IF NOT(xReadFirstTime) THEN
	xReadFirstTime:=TRUE;
END_IF;
(******************************************************************************************************************************************)
(****************************				           Reset Function Part                                                 *****************************)
(******************************************************************************************************************************************)
IF xReset AND NOT(xSetEnd) THEN
	xEnd:=FALSE;
	xSetEnd:=TRUE;
END_IF;
(******************************************************************************************************************************************)
(****************************				              Error Controlling Part                                            *****************************)
(******************************************************************************************************************************************)
xTmp:=	TAxisToolLeft.T_CtrleSingle.xErr OR
		(TAxisToolCenter.T_CtrleSingle.xErr AND xMicroRodActive) OR
		TAxisToolRight.T_CtrleSingle.xErr OR
		TAxisToolFeeder.T_CtrleSingle.xErr OR
		TAxisGrindFeeder.T_CtrleSingle.xErr;
xTmp1:=	NOT(TAxisToolLeft.T_CtrleSingle.xExecute) AND
		((NOT(TAxisToolCenter.T_CtrleSingle.xExecute) AND xMicroRodActive) OR NOT(xMicroRodActive)) AND
		 NOT(TAxisToolRight.T_CtrleSingle.xExecute) AND
		((NOT(TAxisToolFeeder.T_CtrleSingle.xExecute) AND NOT(xMicroRodActive)) OR xMicroRodActive) AND
		NOT(TAxisGrindFeeder.T_CtrleSingle.xExecute);
IF (xHardwareError OR (xTmp AND xStartMainPrc)) AND NOT(xSetEnd) THEN
	IF xTmp1 THEN
		IF NOT(xInitError) THEN
			iStepError:=100;
			xInitError:=TRUE;
			IF xHardwareError THEN
				iErrorNr:=iTmpErrorNr;
			ELSE
				xHardwareError:=TRUE;	(* Hardware Error *)
			END_IF;
		END_IF;
		CASE iStepError OF
			100:	iStepError:=0;
				xError:=TRUE;
		END_CASE;
		IF xQuitErr THEN
			xSetEnd:=TRUE;
		END_IF;
	END_IF;
END_IF;
(******************************************************************************************************************************************)
(****************************				              Main Controlling Part                                            *****************************)
(******************************************************************************************************************************************)
IF (xStart OR xStartMainCtr) AND NOT(xSetEnd) AND NOT(xHardwareError) THEN
	IF NOT (xInitMainCtr) THEN
		iTmpErrorNr:=0;
		iStepPrc:=100;
		xInitMainCtr:=TRUE;
		xStartMainCtr:=TRUE;
		xStart:=FALSE;
		xEnd:=FALSE;
		xAbord:=FALSE;
		xTmpInit:=FALSE;
		xCheckToolFeedPosition:=FALSE;
		xCheckWithoutToolRotation:=FALSE;
		bActivePartNumber:=0;
		lrCalcToolLengthInc:=lrCalcToolLength:=0.0;
		rSpeedToolFeed:=0.0;
	END_IF;
	IF xStop AND NOT(xTmpInit) THEN
		xTmpInit:=TRUE;
		iTmp:=100;
		RETURN;
	END_IF;
	IF xFreeze THEN
		IF xStart AND NOT(xAbord) THEN
			xFreeze:=FALSE;
			xStart:=FALSE;
		END_IF;
		IF xAbord THEN
			xAbord:=FALSE;
			xFreeze:=FALSE;
			xStart:=FALSE;
			xSetEnd:=TRUE;
		END_IF;
		RETURN;
	END_IF;
	IF NOT(xStartMainPrc) AND NOT(xSetEnd) THEN
		xStartMainPrc:=TRUE;
	END_IF;
END_IF;
(******************************************************************************************************************************************)
(****************************		               Controlling of the ToolFeeder Position                            *****************************)
(******************************************************************************************************************************************)
IF xCheckToolFeedPosition THEN
	IF xMicroRodActive THEN
		lrToolFeederPosition:=TAxisToolFeeder.T_LiveValue.lrActualPositionNotModulo - lrSaveToolFeederPosition;
		lrToolFeederActualPosition:=(lrToolFeederPosition / TAxisToolFeeder.T_CtrleSingle.lrScaleFactor);
		lrCalcToolLength:=lrToolFeederActualPosition;
	END_IF;
	IF NOT(xMicroRodActive) AND (TAxisToolRight.T_CtrleSingle.lrGearRatio <> 0.0) THEN
		IF NOT(xCheckWithoutToolRotation) THEN
			lrToolFeedCalcLengthPosition:=((((T_WorkTool.rToolLength * 10.0) / ABS(T_WorkTool.rPitch)) * 24000.0) / TAxisToolRight.T_CtrleSingle.lrScaleFactor);
			lrToolFeederPosition:=lrToolFeederPosition + ABS(ABS(TAxisToolRight.T_LiveValue.lrActualPosition) - (lrSaveToolFeederPosition / TAxisToolRight.T_CtrleSingle.lrScaleFactor));
			lrSaveToolFeederPosition:=ABS(TAxisToolRight.T_LiveValue.lrActualPositionNotModulo);
			lrToolFeederActualPosition:=((T_WorkTool.rToolLength * 10.0) / lrToolFeedCalcLengthPosition) * lrToolFeederPosition;
			lrCalcToolLength:=lrCalcToolLengthInc + lrToolFeederActualPosition;
		ELSE
			lrCalcToolLength:=ABS(TAxisToolFeeder.T_LiveValue.lrActualPosition);
		END_IF;
	END_IF;
ELSE
	xCheckWithoutToolRotation:=FALSE;
	IF NOT(xMicroRodActive) AND (TAxisToolRight.T_CtrleSingle.lrGearRatio <> 0.0) THEN
		lrSaveToolFeederPosition:=ABS(TAxisToolRight.T_LiveValue.lrActualPositionNotModulo);
		lrSaveToolRightPosition:=TAxisToolRight.T_LiveValue.lrActualPositionNotModulo * TAxisToolRight.T_CtrleSingle.lrGearRatio;
		lrCalcToolLengthInc:=lrCalcToolLength;
	END_IF;
	IF xMicroRodActive THEN
		lrSaveToolFeederPosition:=TAxisToolFeeder.T_LiveValue.lrActualPositionNotModulo;
	END_IF;
	lrToolFeederActualPosition:=lrToolFeederPosition:=0.0;
END_IF;
lrProcessToolFeederActualPosition:=lrCalcToolLength;
lrProcessToolFeederSpeed:=rSpeedToolFeed;
(******************************************************************************************************************************************)
(****************************				             immediate Stop Part                                              *****************************)
(******************************************************************************************************************************************)
IF xTmpInit AND NOT(xSetEnd) THEN
	IF NOT(xSafetyCircuitOn) THEN
		xTmpInit:=FALSE;
		iTmp:=100;
		xSetEnd:=TRUE;
		RETURN;
	END_IF;
	CASE iTmp OF
		100:	xReadyToolFeedStop:=xReadyGrindFeedStop:=FALSE;
			TAxisGrindFeeder.T_CtrleSingle.lrAcceleration:=T_Standard.T_TeachINToolFeeder.rAcceleration;
			TAxisGrindFeeder.T_CtrleSingle.lrDecceleration:=T_Standard.T_TeachINToolFeeder.rDeceleration;
			TAxisGrindFeeder.T_CtrleSingle.iFunction:=5;	(* Stop Movement *)
			TAxisGrindFeeder.T_CtrleSingle.xExecute:=TRUE;
			iTmp:=200;
			RETURN;
		200:	IF NOT(TAxisGrindFeeder.T_CtrleSingle.xExecute) AND TAxisGrindFeeder.T_CtrleSingle.xDone THEN
				TAxisGrindFeeder.T_CtrleSingle.lrAcceleration:=T_Standard.T_TeachINGrindFeeder.rAcceleration;
				TAxisGrindFeeder.T_CtrleSingle.lrDecceleration:=T_Standard.T_TeachINGrindFeeder.rDeceleration;
				TAxisGrindFeeder.T_CtrleSingle.lrPosition:=	T_ProcessImageData.T_ProcessPara.rToolDiameterProcess +
														T_ProcessImageData.T_ProcessPara.rSecurityPosGrindFeedProcess;
				TAxisGrindFeeder.T_CtrleSingle.lrVelocity:=T_ProcessImageData.T_ProcessPara.rSpeedBackwardGrindFeed;
				TAxisGrindFeeder.T_CtrleSingle.iFunction:=7;	(* Move Absolut *)
				TAxisGrindFeeder.T_CtrleSingle.xExecute:=TRUE;
				iTmp:=300;
			END_IF;
			RETURN;
		300:	IF NOT(TAxisGrindFeeder.T_CtrleSingle.xExecute) AND TAxisGrindFeeder.T_CtrleSingle.xDone AND NOT(xReadyGrindFeedStop) THEN
				xReadyGrindFeedStop:=TRUE;
			END_IF;
			IF (TAxisGrindFeeder.T_LiveValue.lrActualPosition >= (T_ProcessImageData.T_ProcessPara.rToolDiameterProcess + T_ProcessImageData.T_ProcessPara.rOffsetBeforeToolDiaGrindFeedProcess)) AND NOT(xReadyToolFeedStop) THEN
				xReadyToolFeedStop:=TRUE;
				xCheckToolFeedPosition:=FALSE;
				IF xMicroRodActive THEN
					IF NOT(TAxisToolFeeder.T_CtrleSingle.xNotMoving) THEN
						TAxisToolFeeder.T_CtrleSingle.lrAcceleration:=T_Standard.T_TeachINToolFeeder.rAcceleration;
						TAxisToolFeeder.T_CtrleSingle.lrDecceleration:=T_Standard.T_TeachINToolFeeder.rDeceleration;
						TAxisToolFeeder.T_CtrleSingle.iFunction:=5;	(* Stop Movement *)
						TAxisToolFeeder.T_CtrleSingle.xExecute:=TRUE;
					END_IF;
				END_IF;
				IF NOT(xMicroRodActive) THEN
					FBCalcGearFactor(	rSpeed:= 0.0,
										rToolRotationSpeed:= rToolRotationSpeed,
										T_WorkTool:=T_WorkTool );
					IF (T_WorkTool.rToolRotationSpeed > 0) THEN
						TAxisToolFeeder.T_CtrleSingle.lrGearFactor:=INT_TO_LREAL(FBCalcGearFactor.T_WorkTool.iToolFeederGearFactor) * -1.0;
					ELSE
						TAxisToolFeeder.T_CtrleSingle.lrGearFactor:=INT_TO_LREAL(FBCalcGearFactor.T_WorkTool.iToolFeederGearFactor);
					END_IF;
					TAxisToolFeeder.T_CtrleSingle.lrGearDivider:=INT_TO_LREAL(FBCalcGearFactor.T_WorkTool.iToolFeederGearDivider);
					(* Set Gear Value with PDO Object *)
					TAxisToolFeeder.T_RxPdoParameter.iGearFactor:=LREAL_TO_INT(TAxisToolFeeder.T_CtrleSingle.lrGearFactor);
					TAxisToolFeeder.T_RxPdoParameter.uiGearDivider:=LREAL_TO_UINT(TAxisToolFeeder.T_CtrleSingle.lrGearDivider);
				END_IF;
				lrProcessToolFeederSpeed:=0.0;
			END_IF;
			IF xReadyToolFeedStop AND xReadyGrindFeedStop THEN
				iTmp:=400;
			END_IF;
			RETURN;
		400:	IF NOT(TAxisToolFeeder.T_CtrleSingle.xExecute) AND TAxisToolFeeder.T_CtrleSingle.xDone THEN
				iTmp:=500;
			END_IF;
			RETURN;
		500:	xTmpInit:=FALSE;
			iTmp:=100;
			xSetEnd:=TRUE;
			RETURN;
	END_CASE;
END_IF;
(******************************************************************************************************************************************)
(****************************				             Main Procedure Part                                             *****************************)
(******************************************************************************************************************************************)
IF xStartMainPrc AND NOT(xSetEnd) AND NOT(xHardwareError) THEN
	CASE iStepPrc OF
		(* Initial Procedure *)
		100:	rToolFeedLength:=0.0;
			rToolDiameter:=T_ProcessImageData.T_ProcessPara.rToolDiameterProcess;
			rGrindFeedPlunge:=0.0;
			rSpeedGrindFeed:=0.0;
			rSpeedToolFeed:=0.0;
			iStartSection:=1;
			(* Check Start and End Section of the ToolGeometry *)
			FOR ii:=1 TO 6 DO
				IF T_ProcessImageData.T_GeometryPara.axActiveSection[ii] THEN
					IF (iStartSection = 0) THEN
						iStartSection:=ii;
					END_IF;
					iEndSection:=ii;
				END_IF;
			END_FOR;
			xResetFB:=TRUE;
			FBCalcPlungeGrinding(	rToolDiameter:= T_ProcessImageData.T_ProcessPara.rToolDiameterProcess,
									rToolDiameterWithOffset:=T_ProcessImageData.T_ProcessPara.rToolDiameterProcess + T_ProcessImageData.T_ProcessPara.rOffsetBeforeToolDiaGrindFeedProcess,
									xReset:= xResetFB);
			(* AutoGroove is not aloved to work in more cycle *)
			rPlungeCycleGrindFeedGeometry:=T_ProcessImageData.T_ProcessPara.rToolDiameterProcess;
			xStartMainPrc:=FALSE;
			xInitStep:=FALSE;
(*08.09.2010: KFS	{ *)
(*			iStepPrc:=200;*)
			iStepPrc:=120;
		(* Switch the Axis as Slave for Move ToolRotation to StartPositionGroove*)
		120:	IF NOT(xInitStep) THEN
				xInitStep:=TRUE;
				IF rStartPosAutoGrooveToolRotation<> 0 THEN
					IF NOT(TAxisToolCenter.T_CtrleSingle.xSlave) THEN
						TAxisToolCenter.T_CtrleSingle.lrGearDivider:=INT_TO_LREAL(T_WorkTool.iBaseGearDivider);
						TAxisToolCenter.T_CtrleSingle.lrGearFactor:=(INT_TO_LREAL(T_WorkTool.iBaseGearDivider) /
																				(TAxisToolLeft.T_CtrleSingle.lrGearRatio /
																				TAxisToolCenter.T_CtrleSingle.lrGearRatio) ) * -1.0;
						TAxisToolCenter.T_CtrleSingle.iFunction:=25;
						TAxisToolCenter.T_CtrleSingle.xExecute:=TRUE;
					END_IF;
					IF NOT(TAxisToolRight.T_CtrleSingle.xSlave) THEN
						TAxisToolRight.T_CtrleSingle.lrGearDivider:=INT_TO_LREAL(T_WorkTool.iBaseGearDivider);
						TAxisToolRight.T_CtrleSingle.lrGearFactor:=	INT_TO_LREAL(T_WorkTool.iBaseGearDivider) /
																				(TAxisToolLeft.T_CtrleSingle.lrGearRatio /
																				TAxisToolRight.T_CtrleSingle.lrGearRatio);
						TAxisToolRight.T_CtrleSingle.iFunction:=25;
						TAxisToolRight.T_CtrleSingle.xExecute:=TRUE;
					END_IF;
				END_IF;
			END_IF;
			IF NOT(TAxisToolCenter.T_CtrleSingle.xExecute) AND TAxisToolCenter.T_CtrleSingle.xDone  AND
			    NOT(TAxisToolRight.T_CtrleSingle.xExecute) AND TAxisToolRight.T_CtrleSingle.xDone  THEN
				xStartMainPrc:=FALSE;
				xInitStep:=FALSE;
				iStepPrc:=150;
			END_IF
		(*Rotate Tool to the StartPositionGroove*)
		150:IF NOT(xInitStep) THEN
				xInitStep:=TRUE;
				IF rStartPosAutoGrooveToolRotation<> 0 THEN
					lrSavePos:=TAxisToolLeft.T_LiveValue.lrActualPositionRelativ;
					TAxisToolLeft.T_CtrleSingle.lrDistance:= rStartPosAutoGrooveToolRotation;
					TAxisToolLeft.T_CtrleSingle.lrVelocity:=T_WorkTool.rToolRotationSpeed;
					TAxisToolLeft.T_CtrleSingle.iFunction:=8;
					TAxisToolLeft.T_CtrleSingle.xExecute:=TRUE;
				END_IF;
			END_IF;
			IF NOT(TAxisToolLeft.T_CtrleSingle.xExecute) AND TAxisToolLeft.T_CtrleSingle.xDone THEN
				xStartMainPrc:=FALSE;
				xInitStep:=FALSE;
				iStepPrc:=200;
			END_IF;
(*08.09.2010: KFS	} *)
		(* Calculation first only for the Plunge Procedure *)
		200:	IF NOT(xInitStep) THEN
				xInitStep:=TRUE;
				FBCalcPlungeGrinding(	T_Geometry:= T_ProcessImageData.T_GeometryPara,
										T_AutoGeometryPara:= T_ProcessImageData.T_AutoGeometryPara,
										rToolDiameter:= T_ProcessImageData.T_ProcessPara.rToolDiameterProcess,
										rToolDiameterWithOffset:=T_ProcessImageData.T_ProcessPara.rToolDiameterProcess + T_ProcessImageData.T_ProcessPara.rOffsetBeforeToolDiaGrindFeedProcess,
										rPlungeCycleGrindFeedGeometry:=rPlungeCycleGrindFeedGeometry,
										iStartSection:= iStartSection,
										iEndSection:= iEndSection,
										xReset:= xResetFB);
			END_IF;
			IF xInitStep THEN
				bActivePartNumber:=INT_TO_BYTE(FBCalcPlungeGrinding.iStepSectionWork);
				xStartMainPrc:=FALSE;
				xInitStep:=FALSE;
				IF xDoNotMoveGrindPosition THEN
					iStepPrc:=500;
				ELSE
					iStepPrc:=300;
				END_IF;
			END_IF;
		(* start with the plunge procedure *)
		300:	IF NOT(xInitStep) THEN
				xInitStep:=TRUE;
				rToolFeedLength:=0.0;
				rSpeedToolFeed:=0.0;
				IF T_ProcessImageData.T_AutoGroovePara.xPlungeActivationGroove THEN
					rToolFeedLength:=T_ProcessImageData.T_AutoGroovePara.rPlungeLengthToolFeedGroove;
					T_WorkTool.rToolLength:=rToolFeedLength/10.0;
				ELSE
					T_WorkTool.rToolLength:=0.0;
				END_IF;
				IF T_ProcessImageData.T_AutoGroovePara.xPlungeActivationGroove THEN
					T_WorkTool.rToolRotationSpeed:=T_ProcessImageData.T_AutoGroovePara.rSpeedToolRotationGroove;
					T_WorkTool.rPitch:=T_ProcessImageData.T_AutoGroovePara.rPitchGroove * -1.0;
					T_WorkTool.rGrindFeederPlunge:=	FBCalcPlungeGrinding.rGrindingRelativePosition;
					FBToolCalcul(	xMicroRodActive:=xMicroRodActive,
									xBeckhoffDriveActive:=FALSE,
									T_WorkTool:= T_WorkTool,
									rToolFeedAcclDecl:= T_Standard.T_TeachINToolFeeder.rAcceleration);
					rGrindFeedPlunge:=T_WorkTool.rGrindFeederPlunge * -1.0;
					rSpeedGrindFeed:=T_WorkTool.rGrindFeederSpeedUnit;
					rSpeedToolFeed:=T_WorkTool.rToolFeederSpeedUnit * -1.0;
				ELSE
					rSpeedGrindFeed:=T_ProcessImageData.T_AutoGroovePara.rPlungeSpeedGrindFeedGroove;
					rGrindFeedPlunge:=FBCalcPlungeGrinding.rGrindingRelativePosition * -1.0;
					IF (rToolFeedLength <> 0) THEN
						rTimeGrindPlunge:=ABS(rGrindFeedPlunge) / rSpeedGrindFeed;		(* calc Time in seocnds *)
						rSpeedToolFeed:=rToolFeedLength / rTimeGrindPlunge;	(* calc Speed ToolFeed in mm/s *)
					END_IF;
					T_WorkTool.rPitch:=T_ProcessImageData.T_AutoGroovePara.rPitchGroove * -1.0;
				END_IF;
				rToolRotationSpeed:=T_ProcessImageData.T_AutoGroovePara.rSpeedToolRotationGroove;
				(* Start Relative movement of the GrindAxis *)
				TAxisGrindFeeder.T_CtrleSingle.lrAcceleration:=T_Standard.T_TeachINGrindFeeder.rAcceleration;
				TAxisGrindFeeder.T_CtrleSingle.lrDecceleration:=T_Standard.T_TeachINGrindFeeder.rDeceleration;
				TAxisGrindFeeder.T_CtrleSingle.lrDistance:=rGrindFeedPlunge;
				TAxisGrindFeeder.T_CtrleSingle.lrVelocity:=rSpeedGrindFeed;
				TAxisGrindFeeder.T_CtrleSingle.iFunction:=8;	(* Move Relative *)
				TAxisGrindFeeder.T_CtrleSingle.xExecute:=TRUE;
				IF (rToolFeedLength <> 0) THEN
					xCheckToolFeedPosition:=TRUE;	(* Start Measure Relative Position of the ToolFeeder *)
					xCheckWithoutToolRotation:=TRUE;
					(* Start continuos movement of the ToolFeeder Axis *)
					TAxisToolFeeder.T_CtrleSingle.lrAcceleration:=T_Standard.T_TeachINToolFeeder.rAcceleration;
					TAxisToolFeeder.T_CtrleSingle.lrDecceleration:=T_Standard.T_TeachINToolFeeder.rDeceleration;
					TAxisToolFeeder.T_CtrleSingle.lrVelocity:=rSpeedToolFeed;
					TAxisToolFeeder.T_CtrleSingle.iFunction:=6;	(* Move continue velocity *)
					TAxisToolFeeder.T_CtrleSingle.xExecute:=TRUE;
				END_IF;
			END_IF;
			IF NOT(TAxisGrindFeeder.T_CtrleSingle.xExecute) AND TAxisGrindFeeder.T_CtrleSingle.xDone THEN
				xCheckToolFeedPosition:=FALSE;
				xCheckWithoutToolRotation:=FALSE;
				xStartMainPrc:=FALSE;
				xInitStep:=FALSE;
				IF (rToolFeedLength <> 0) THEN
					iStepPrc:=400;
				ELSE
					iStepPrc:=600;
				END_IF;
			END_IF;
		(* Stop the movement of the ToolFeeder *)
		400:	IF NOT(xInitStep) THEN
				xInitStep:=TRUE;
				TAxisToolFeeder.T_CtrleSingle.lrAcceleration:=T_Standard.T_TeachINToolFeeder.rAcceleration;
				TAxisToolFeeder.T_CtrleSingle.lrDecceleration:=T_Standard.T_TeachINToolFeeder.rDeceleration;
				TAxisToolFeeder.T_CtrleSingle.iFunction:=5;	(* Stop Movement *)
				TAxisToolFeeder.T_CtrleSingle.xExecute:=TRUE;
			END_IF;
			IF NOT(TAxisToolFeeder.T_CtrleSingle.xExecute) AND TAxisToolFeeder.T_CtrleSingle.xDone THEN
				xStartMainPrc:=FALSE;
				xInitStep:=FALSE;
				 iStepPrc:=600;
			END_IF;
		(* Override the Position of the GrindFeeder Axis with the Diameter of the first working section *)
		500:IF NOT(xInitStep) THEN
				xInitStep:=TRUE;
				TAxisGrindFeeder.T_CtrleSingle.rSetPosition:=T_ProcessImageData.T_GeometryPara.arStartDiameter[iStartSection];
				TAxisGrindFeeder.T_CtrleSingle.iFunction:=11;
				TAxisGrindFeeder.T_CtrleSingle.xExecute:=TRUE;
			END_IF;
			IF NOT(TAxisGrindFeeder.T_CtrleSingle.xExecute) AND TAxisGrindFeeder.T_CtrleSingle.xDone THEN
				xStartMainPrc:=FALSE;
				xInitStep:=FALSE;
			END_IF;
		(* Switch the Axis as Slave *)
		600:IF NOT(xInitStep) THEN
				xInitStep:=TRUE;
				FBCalcPlungeGrinding(	T_Geometry:= T_ProcessImageData.T_GeometryPara,
										T_AutoGeometryPara:= T_ProcessImageData.T_AutoGeometryPara,
										rToolDiameter:= T_ProcessImageData.T_ProcessPara.rToolDiameterProcess,
										rToolDiameterWithOffset:=T_ProcessImageData.T_ProcessPara.rToolDiameterProcess + T_ProcessImageData.T_ProcessPara.rOffsetBeforeToolDiaGrindFeedProcess,
										rPlungeCycleGrindFeedGeometry:=rPlungeCycleGrindFeedGeometry,
										iStartSection:= iStartSection,
										iEndSection:= iEndSection,
										xReset:= xResetFB);
				(* Check first active section *)
				bActivePartNumber:=INT_TO_BYTE(FBCalcPlungeGrinding.iStepSectionWork);
				iTmpStartSection:=iStartSection + (FBCalcPlungeGrinding.iStepSectionWork - 1);
				T_WorkTool.rToolRotationSpeed:=T_ProcessImageData.T_AutoGroovePara.rSpeedToolRotationGroove;
				T_WorkTool.rPitch:=T_ProcessImageData.T_AutoGroovePara.rPitchGroove * -1.0;
				T_WorkTool.rToolLength:=T_ProcessImageData.T_GeometryPara.arSectionLength[iTmpStartSection];
				rGrindFeedPlunge:=FBCalcPlungeGrinding.rGrindingRelativePosition * -1.0;
				T_WorkTool.rGrindFeederPlunge:=rGrindFeedPlunge;
				FBToolCalcul(	xMicroRodActive:=xMicroRodActive,
								xBeckhoffDriveActive:=FALSE,
								T_WorkTool:= T_WorkTool,
								rToolFeedAcclDecl:= 0.0	);
				rSpeedGrindFeed:=T_WorkTool.rGrindFeederSpeedUnit;
				rToolFeedLength:=T_WorkTool.rToolLength;
				rSpeedToolFeed:=T_WorkTool.rToolFeederSpeedUnit;
				rToolRotationSpeed:=T_WorkTool.rToolRotationSpeed;
				IF xMicroRodActive THEN
					IF NOT(TAxisToolCenter.T_CtrleSingle.xSlave) THEN
						TAxisToolCenter.T_CtrleSingle.lrGearDivider:=INT_TO_LREAL(T_WorkTool.iBaseGearDivider);
						TAxisToolCenter.T_CtrleSingle.lrGearFactor:=(INT_TO_LREAL(T_WorkTool.iBaseGearDivider) /
																				(TAxisToolLeft.T_CtrleSingle.lrGearRatio /
																				TAxisToolCenter.T_CtrleSingle.lrGearRatio) ) * -1.0;
						TAxisToolCenter.T_CtrleSingle.iFunction:=25;
						TAxisToolCenter.T_CtrleSingle.xExecute:=TRUE;
					END_IF;
					IF NOT(TAxisToolRight.T_CtrleSingle.xSlave) THEN
						TAxisToolRight.T_CtrleSingle.lrGearDivider:=INT_TO_LREAL(T_WorkTool.iBaseGearDivider);
						TAxisToolRight.T_CtrleSingle.lrGearFactor:=	INT_TO_LREAL(T_WorkTool.iBaseGearDivider) /
																				(TAxisToolLeft.T_CtrleSingle.lrGearRatio /
																				TAxisToolRight.T_CtrleSingle.lrGearRatio);
						TAxisToolRight.T_CtrleSingle.iFunction:=25;
						TAxisToolRight.T_CtrleSingle.xExecute:=TRUE;
					END_IF;
				END_IF;
				IF NOT xMicroRodActive THEN
					IF NOT(TAxisToolRight.T_CtrleSingle.xSlave) THEN
						TAxisToolRight.T_CtrleSingle.lrGearDivider:=INT_TO_LREAL(T_WorkTool.iBaseGearDivider);
						TAxisToolRight.T_CtrleSingle.lrGearFactor:=	(INT_TO_LREAL(T_WorkTool.iBaseGearDivider) /
																				(TAxisToolLeft.T_CtrleSingle.lrGearRatio /
																				TAxisToolRight.T_CtrleSingle.lrGearRatio)) * -1.0;
						TAxisToolRight.T_CtrleSingle.iFunction:=25;
						TAxisToolRight.T_CtrleSingle.xExecute:=TRUE;
					END_IF;
				END_IF;
				IF NOT(TAxisToolFeeder.T_CtrleSingle.xSlave) THEN
					IF (T_WorkTool.rToolRotationSpeed > 0) THEN
						TAxisToolFeeder.T_CtrleSingle.lrGearFactor:=INT_TO_LREAL(T_WorkTool.iToolFeederGearFactor) * -1.0;
					ELSE
						TAxisToolFeeder.T_CtrleSingle.lrGearFactor:=INT_TO_LREAL(T_WorkTool.iToolFeederGearFactor);
					END_IF;
					TAxisToolFeeder.T_CtrleSingle.lrGearDivider:=INT_TO_LREAL(T_WorkTool.iToolFeederGearDivider);
					(* Set Gear Value with PDO Object *)
					TAxisToolFeeder.T_RxPdoParameter.iGearFactor:=LREAL_TO_INT(TAxisToolFeeder.T_CtrleSingle.lrGearFactor);
					TAxisToolFeeder.T_RxPdoParameter.uiGearDivider:=LREAL_TO_UINT(TAxisToolFeeder.T_CtrleSingle.lrGearDivider);
					TAxisToolFeeder.T_CtrleSingle.iFunction:=25;
					TAxisToolFeeder.T_CtrleSingle.xExecute:=TRUE;
				END_IF;
			END_IF;
			IF ((NOT(TAxisToolCenter.T_CtrleSingle.xExecute) AND TAxisToolCenter.T_CtrleSingle.xDone AND xMicroRodActive) OR NOT(xMicroRodActive)) AND
			    NOT(TAxisToolRight.T_CtrleSingle.xExecute) AND TAxisToolRight.T_CtrleSingle.xDone AND
			    ((NOT(TAxisToolFeeder.T_CtrleSingle.xExecute) AND TAxisToolFeeder.T_CtrleSingle.xDone AND NOT(xMicroRodActive)) OR xMicroRodActive) THEN
				xStartMainPrc:=FALSE;
				xInitStep:=FALSE;
				iStepPrc:=700;
			END_IF;
		(* Start ToolRotation and the ToolFeeder as Slave from the ToolRotation and the Grinding if it work a cone Section *)
		700:IF NOT(xInitStep) THEN
				xInitStep:=TRUE;
				(* Start ToolRotation *)
				TAxisToolLeft.T_CtrleSingle.lrVelocity:=T_WorkTool.rToolRotationSpeed;
				TAxisToolLeft.T_CtrleSingle.iFunction:=6;
				TAxisToolLeft.T_CtrleSingle.xExecute:=TRUE;
				(*Check if it work a Cone section*)
				IF (rGrindFeedPlunge <> 0) THEN
					xGrindFeedMaster:=TRUE;
					xCheckToolFeedPosition:=TRUE;	(* Start Measure Relative Position of the ToolFeeder *)
					IF (TAxisGrindFeeder.T_CtrleSingle.iFunction <> 11) THEN
						TAxisGrindFeeder.T_CtrleSingle.xBlockAcclDeclParameter:=TRUE;	(* do not send again the accl and decl parameter-->better performance *)
					END_IF;
					TAxisGrindFeeder.T_CtrleSingle.lrAcceleration:=T_Standard.T_TeachINGrindFeeder.rAcceleration;
					TAxisGrindFeeder.T_CtrleSingle.lrDecceleration:=T_Standard.T_TeachINGrindFeeder.rDeceleration;
					TAxisGrindFeeder.T_CtrleSingle.lrDistance:=rGrindFeedPlunge;
					TAxisGrindFeeder.T_CtrleSingle.lrVelocity:=rSpeedGrindFeed;
					TAxisGrindFeeder.T_CtrleSingle.iFunction:=8;	(* Move Relative *)
					TAxisGrindFeeder.T_CtrleSingle.xExecute:=TRUE;
				ELSE
					xGrindFeedMaster:=FALSE;
					xCheckToolFeedPosition:=TRUE;	(* Start Measure Relative Position of the ToolFeeder *)
				END_IF;
			END_IF;
			IF xGrindFeedMaster THEN
				(* This is active by work a cone section *)
				IF (NOT(TAxisGrindFeeder.T_CtrleSingle.xExecute) AND TAxisGrindFeeder.T_CtrleSingle.xDone) THEN
					xCheckToolFeedPosition:=FALSE;
					xStartMainPrc:=FALSE;
					xInitStep:=FALSE;
					iStepPrc:=800;
				END_IF;
			END_IF;
			IF NOT(xGrindFeedMaster) THEN
				(* This is only active if it is work a cylinder section *)
				IF (lrToolFeederActualPosition > (rToolFeedLength * 10.0)) THEN
					xCheckToolFeedPosition:=FALSE;
					xStartMainPrc:=FALSE;
					xInitStep:=FALSE;
					iStepPrc:=800;
				END_IF;
			END_IF;
		(* Init the next Section *)
		800:IF NOT(xInitStep) THEN
				xInitStep:=TRUE;
				FBCalcPlungeGrinding(	T_Geometry:= T_ProcessImageData.T_GeometryPara,
										T_AutoGeometryPara:= T_ProcessImageData.T_AutoGeometryPara,
										rToolDiameter:= T_ProcessImageData.T_ProcessPara.rToolDiameterProcess,
										rToolDiameterWithOffset:=T_ProcessImageData.T_ProcessPara.rToolDiameterProcess + T_ProcessImageData.T_ProcessPara.rOffsetBeforeToolDiaGrindFeedProcess,
										rPlungeCycleGrindFeedGeometry:=rPlungeCycleGrindFeedGeometry,
										iStartSection:= iStartSection,
										iEndSection:= iEndSection,
										xReset:= xResetFB);
				(* Check first active section *)
				bActivePartNumber:=INT_TO_BYTE(FBCalcPlungeGrinding.iStepSectionWork);
				iTmpStartSection:=iStartSection + (FBCalcPlungeGrinding.iStepSectionWork - 1);
				T_WorkTool.rToolRotationSpeed:=T_ProcessImageData.T_AutoGroovePara.rSpeedToolRotationGroove;
				T_WorkTool.rPitch:=T_ProcessImageData.T_AutoGroovePara.rPitchGroove * -1.0;
				T_WorkTool.rToolLength:=T_ProcessImageData.T_GeometryPara.arSectionLength[iTmpStartSection];
				rGrindFeedPlunge:=FBCalcPlungeGrinding.rGrindingRelativePosition * -1.0;
				T_WorkTool.rGrindFeederPlunge:=rGrindFeedPlunge;
				FBToolCalcul(	xMicroRodActive:=xMicroRodActive,
								xBeckhoffDriveActive:=FALSE,
								T_WorkTool:= T_WorkTool,
								rToolFeedAcclDecl:= 0.0	);
				rSpeedGrindFeed:=T_WorkTool.rGrindFeederSpeedUnit;
				rToolFeedLength:=T_WorkTool.rToolLength;
				rSpeedToolFeed:=T_WorkTool.rToolFeederSpeedUnit;
				rToolRotationSpeed:=T_WorkTool.rToolRotationSpeed;
			END_IF;
			IF xInitStep THEN
				xStartMainPrc:=FALSE;
				xInitStep:=FALSE;
				IF (FBCalcPlungeGrinding.iStepSectionWork <> 7) THEN
					iStepPrc:=900;	(* Work the Geometry Section *)
				ELSE
					iStepPrc:=1000;	(* Work the Displace Procedure *)
				END_IF;
			END_IF;
		(* Work the next Section *)
		900:IF NOT(xInitStep) THEN
				xInitStep:=TRUE;
				(*Check if it work a Cone section*)
				IF (rGrindFeedPlunge <> 0) THEN
					xGrindFeedMaster:=TRUE;
					xCheckToolFeedPosition:=TRUE;	(* Start Measure Relative Position of the ToolFeeder *)
					TAxisGrindFeeder.T_CtrleSingle.xBlockAcclDeclParameter:=TRUE;	(* do not send again the accl and decl parameter-->better performance *)
					TAxisGrindFeeder.T_CtrleSingle.lrAcceleration:=T_Standard.T_TeachINGrindFeeder.rAcceleration;
					TAxisGrindFeeder.T_CtrleSingle.lrDecceleration:=T_Standard.T_TeachINGrindFeeder.rDeceleration;
					TAxisGrindFeeder.T_CtrleSingle.lrDistance:=rGrindFeedPlunge;
					TAxisGrindFeeder.T_CtrleSingle.lrVelocity:=rSpeedGrindFeed;
					TAxisGrindFeeder.T_CtrleSingle.iFunction:=8;	(* Move Relative *)
					TAxisGrindFeeder.T_CtrleSingle.xExecute:=TRUE;
				ELSE
					xGrindFeedMaster:=FALSE;
					xCheckToolFeedPosition:=TRUE;	(* Start Measure Relative Position of the ToolFeeder *)
					IF NOT(xMicroRodActive) THEN
						IF (T_WorkTool.rToolRotationSpeed > 0) THEN
							TAxisToolFeeder.T_CtrleSingle.lrGearFactor:=INT_TO_LREAL(T_WorkTool.iToolFeederGearFactor) * -1.0;
						ELSE
							TAxisToolFeeder.T_CtrleSingle.lrGearFactor:=INT_TO_LREAL(T_WorkTool.iToolFeederGearFactor);
						END_IF;
						TAxisToolFeeder.T_CtrleSingle.lrGearDivider:=INT_TO_LREAL(T_WorkTool.iToolFeederGearDivider);
						(* Set Gear Value with PDO Object *)
						TAxisToolFeeder.T_RxPdoParameter.iGearFactor:=LREAL_TO_INT(TAxisToolFeeder.T_CtrleSingle.lrGearFactor);
						TAxisToolFeeder.T_RxPdoParameter.uiGearDivider:=LREAL_TO_UINT(TAxisToolFeeder.T_CtrleSingle.lrGearDivider);
					END_IF;
				END_IF;
			END_IF;
			IF xGrindFeedMaster THEN
				(* This is active by work a cone section *)
				IF (NOT(TAxisGrindFeeder.T_CtrleSingle.xExecute) AND TAxisGrindFeeder.T_CtrleSingle.xDone) THEN
					xCheckToolFeedPosition:=FALSE;
					xStartMainPrc:=FALSE;
					xInitStep:=FALSE;
					iStepPrc:=800;
				END_IF;
			END_IF;
			IF NOT(xGrindFeedMaster) THEN
				(* This is only active if it is work a cylinder section *)
				IF (lrToolFeederActualPosition > (rToolFeedLength * 10.0)) THEN
					xCheckToolFeedPosition:=FALSE;
					xStartMainPrc:=FALSE;
					xInitStep:=FALSE;
					iStepPrc:=800;
				END_IF;
			END_IF;
		(* start with the displace procedure *)
		1000:IF NOT(xInitStep) THEN
				xInitStep:=TRUE;
				rToolFeedLength:=0.0;
				rSpeedToolFeed:=0.0;
				IF T_ProcessImageData.T_AutoGroovePara.xDisplaceActivationGroove THEN
					rToolFeedLength:=T_ProcessImageData.T_AutoGroovePara.rDisplaceLengthToolFeedGroove;
					T_WorkTool.rToolLength:=rToolFeedLength/10.0;
				ELSE
					T_WorkTool.rToolLength:=0.0;
				END_IF;
				IF T_ProcessImageData.T_AutoGroovePara.xDisplaceActivationGroove THEN
					T_WorkTool.rToolRotationSpeed:=T_ProcessImageData.T_AutoGroovePara.rSpeedToolRotationGroove;
					T_WorkTool.rPitch:=T_ProcessImageData.T_AutoGroovePara.rPitchGroove * -1.0;
					T_WorkTool.rGrindFeederPlunge:=	FBCalcPlungeGrinding.rGrindingRelativePosition * -1.0;
					FBToolCalcul(	xMicroRodActive:=xMicroRodActive,
								  	xBeckhoffDriveActive:=FALSE,
								  	T_WorkTool:= T_WorkTool,
								  	rToolFeedAcclDecl:= T_Standard.T_TeachINToolFeeder.rDeceleration	);
					rGrindFeedPlunge:=T_WorkTool.rGrindFeederPlunge;
					rSpeedGrindFeed:=T_WorkTool.rGrindFeederSpeedUnit;
					rSpeedToolFeed:=T_WorkTool.rToolFeederSpeedUnit * -1.0;
				ELSE
					rSpeedGrindFeed:=T_ProcessImageData.T_AutoGroovePara.rDisplaceSpeedGrindFeedGroove;
					rGrindFeedPlunge:=FBCalcPlungeGrinding.rGrindingRelativePosition * -1.0;
					IF (rToolFeedLength <> 0) THEN
						rTimeGrindPlunge:=ABS(rGrindFeedPlunge) / rSpeedGrindFeed;		(* calc Time in seocnds *)
						rSpeedToolFeed:=(rToolFeedLength * 10.0) / rTimeGrindPlunge;	(* calc Speed ToolFeed in mm/s *)
					END_IF;
					T_WorkTool.rPitch:=T_ProcessImageData.T_AutoGroovePara.rPitchGroove * -1.0;
				END_IF;
				rToolRotationSpeed:=T_ProcessImageData.T_AutoGroovePara.rSpeedToolRotationGroove;
				(* Start Relative movement of the GrindAxis *)
				TAxisGrindFeeder.T_CtrleSingle.xBlockAcclDeclParameter:=TRUE;	(* do not send again the accl and decl parameter-->better performance *)
				TAxisGrindFeeder.T_CtrleSingle.lrAcceleration:=T_Standard.T_TeachINGrindFeeder.rAcceleration;
				TAxisGrindFeeder.T_CtrleSingle.lrDecceleration:=T_Standard.T_TeachINGrindFeeder.rDeceleration;
				TAxisGrindFeeder.T_CtrleSingle.lrDistance:=rGrindFeedPlunge;
				TAxisGrindFeeder.T_CtrleSingle.lrVelocity:=rSpeedGrindFeed;
				TAxisGrindFeeder.T_CtrleSingle.iFunction:=8;	(* Move Relative *)
				TAxisGrindFeeder.T_CtrleSingle.xExecute:=TRUE;
				IF (rToolFeedLength = 0) THEN
				(* Stop ToolFeeder Movement *)
					IF xMicroRodActive THEN
						(* All rotation axis stop since they are the slave of the left axis*)
						TAxisToolLeft.T_CtrleSingle.iFunction:=5;
						TAxisToolLeft.T_CtrleSingle.xExecute:=TRUE;
						IF TAxisToolFeeder.T_CtrleSingle.xSlave THEN
							IF (T_WorkTool.rToolRotationSpeed > 0) THEN
								TAxisToolFeeder.T_CtrleSingle.lrGearFactor:=INT_TO_LREAL(T_WorkTool.iBaseGearDivider) * -1.0;
							ELSE
								TAxisToolFeeder.T_CtrleSingle.lrGearFactor:=INT_TO_LREAL(T_WorkTool.iBaseGearDivider);
							END_IF;
							TAxisToolFeeder.T_CtrleSingle.lrGearDivider:=INT_TO_LREAL(T_WorkTool.iBaseGearDivider);
							(* Set Gear Value with PDO Object *)
							TAxisToolFeeder.T_RxPdoParameter.iGearFactor:=(LREAL_TO_INT(TAxisToolFeeder.T_CtrleSingle.lrGearFactor) * -1);
							TAxisToolFeeder.T_RxPdoParameter.uiGearDivider:=LREAL_TO_UINT(TAxisToolFeeder.T_CtrleSingle.lrGearDivider);
							TAxisToolFeeder.T_CtrleSingle.iFunction:=25;
							TAxisToolFeeder.T_CtrleSingle.xExecute:=TRUE;
						END_IF;
					END_IF;
					IF NOT(xMicroRodActive) THEN
						FBCalcGearFactor(	rSpeed:= 0.0,
											rToolRotationSpeed:= rToolRotationSpeed,
											T_WorkTool:=T_WorkTool );
						IF (T_WorkTool.rToolRotationSpeed > 0) THEN
							TAxisToolFeeder.T_CtrleSingle.lrGearFactor:=INT_TO_LREAL(FBCalcGearFactor.T_WorkTool.iToolFeederGearFactor) * -1.0;
						ELSE
							TAxisToolFeeder.T_CtrleSingle.lrGearFactor:=INT_TO_LREAL(FBCalcGearFactor.T_WorkTool.iToolFeederGearFactor);
						END_IF;
						TAxisToolFeeder.T_CtrleSingle.lrGearDivider:=INT_TO_LREAL(FBCalcGearFactor.T_WorkTool.iToolFeederGearDivider);
						(* Set Gear Value with PDO Object *)
						TAxisToolFeeder.T_RxPdoParameter.iGearFactor:=LREAL_TO_INT(TAxisToolFeeder.T_CtrleSingle.lrGearFactor);
						TAxisToolFeeder.T_RxPdoParameter.uiGearDivider:=LREAL_TO_UINT(TAxisToolFeeder.T_CtrleSingle.lrGearDivider);
					END_IF;
				ELSE
					xCheckToolFeedPosition:=TRUE;	(* Start Measure Relative Position of the ToolFeeder *)
				END_IF;
			END_IF;
			IF NOT(TAxisGrindFeeder.T_CtrleSingle.xExecute) AND TAxisGrindFeeder.T_CtrleSingle.xDone THEN
				xStartMainPrc:=FALSE;
				xInitStep:=FALSE;
				iStepPrc:=1100;
			END_IF;
		(* Check if ToolFeeder Moves and stop it if it moves *)
		1100:IF NOT(xInitStep) THEN
				xInitStep:=TRUE;
				xCheckToolFeedPosition:=FALSE;
				IF xMicroRodActive THEN
					(* All rotation axis stop since they are the slave of the left axis*)
					TAxisToolLeft.T_CtrleSingle.iFunction:=5;
					TAxisToolLeft.T_CtrleSingle.xExecute:=TRUE;
					IF TAxisToolFeeder.T_CtrleSingle.xSlave THEN
						IF (T_WorkTool.rToolRotationSpeed > 0) THEN
							TAxisToolFeeder.T_CtrleSingle.lrGearFactor:=INT_TO_LREAL(T_WorkTool.iBaseGearDivider) * -1.0;
						ELSE
							TAxisToolFeeder.T_CtrleSingle.lrGearFactor:=INT_TO_LREAL(T_WorkTool.iBaseGearDivider);
						END_IF;
						TAxisToolFeeder.T_CtrleSingle.lrGearDivider:=INT_TO_LREAL(T_WorkTool.iBaseGearDivider);
						(* Set Gear Value with PDO Object *)
						TAxisToolFeeder.T_RxPdoParameter.iGearFactor:=(LREAL_TO_INT(TAxisToolFeeder.T_CtrleSingle.lrGearFactor) * -1);
						TAxisToolFeeder.T_RxPdoParameter.uiGearDivider:=LREAL_TO_UINT(TAxisToolFeeder.T_CtrleSingle.lrGearDivider);
						TAxisToolFeeder.T_CtrleSingle.iFunction:=25;
						TAxisToolFeeder.T_CtrleSingle.xExecute:=TRUE;
					END_IF;
				END_IF;
				IF NOT(xMicroRodActive) THEN
					FBCalcGearFactor(	rSpeed:= 0.0,
										rToolRotationSpeed:= rToolRotationSpeed,
										T_WorkTool:=T_WorkTool );
					IF (T_WorkTool.rToolRotationSpeed > 0) THEN
						TAxisToolFeeder.T_CtrleSingle.lrGearFactor:=INT_TO_LREAL(FBCalcGearFactor.T_WorkTool.iToolFeederGearFactor) * -1.0;
					ELSE
						TAxisToolFeeder.T_CtrleSingle.lrGearFactor:=INT_TO_LREAL(FBCalcGearFactor.T_WorkTool.iToolFeederGearFactor);
					END_IF;
					TAxisToolFeeder.T_CtrleSingle.lrGearDivider:=INT_TO_LREAL(FBCalcGearFactor.T_WorkTool.iToolFeederGearDivider);
					(* Set Gear Value with PDO Object *)
					TAxisToolFeeder.T_RxPdoParameter.iGearFactor:=LREAL_TO_INT(TAxisToolFeeder.T_CtrleSingle.lrGearFactor);
					TAxisToolFeeder.T_RxPdoParameter.uiGearDivider:=LREAL_TO_UINT(TAxisToolFeeder.T_CtrleSingle.lrGearDivider);
				END_IF;
			END_IF;
			IF NOT(TAxisToolFeeder.T_CtrleSingle.xExecute) AND TAxisToolFeeder.T_CtrleSingle.xDone THEN
				xStartMainPrc:=FALSE;
				xInitStep:=FALSE;
				iStepPrc:=1200;
			END_IF;
		(* GrindFeeder go to Security Position *)
		1200:IF NOT(xInitStep) THEN
				xInitStep:=TRUE;
				TAxisGrindFeeder.T_CtrleSingle.lrAcceleration:=T_Standard.T_TeachINGrindFeeder.rAcceleration;
				TAxisGrindFeeder.T_CtrleSingle.lrDecceleration:=T_Standard.T_TeachINGrindFeeder.rDeceleration;
				TAxisGrindFeeder.T_CtrleSingle.lrPosition:=	T_ProcessImageData.T_ProcessPara.rToolDiameterProcess +
														T_ProcessImageData.T_ProcessPara.rSecurityPosGrindFeedProcess;
				TAxisGrindFeeder.T_CtrleSingle.lrVelocity:=T_ProcessImageData.T_ProcessPara.rSpeedBackwardGrindFeed;
				TAxisGrindFeeder.T_CtrleSingle.iFunction:=7;	(* Move Absolut *)
				TAxisGrindFeeder.T_CtrleSingle.xExecute:=TRUE;
			END_IF;
			IF NOT(TAxisGrindFeeder.T_CtrleSingle.xExecute) AND TAxisGrindFeeder.T_CtrleSingle.xDone THEN
				(* Procedure is finished *)
				xStartMainPrc:=FALSE;
				xInitStep:=FALSE;
				iStepPrc:=0;
				xSetEnd:=TRUE;
			END_IF;
	END_CASE;
END_IF;
(******************************************************************************************************************************************)
(****************************				           Parallel Procedure Part                                          *****************************)
(******************************************************************************************************************************************)
(******************************************************************************************************************************************)
(****************************				             	Init / Reset Part                                                   *****************************)
(******************************************************************************************************************************************)
IF xSetEnd THEN
	xEnd:=TRUE;
	xInitStep:=FALSE;
	xSetEnd:=FALSE;
	xStop:=FALSE;
	xStartMainPrc:=FALSE;
	xInitMainCtr:=FALSE;
	xStartMainCtr:=FALSE;
	xStart:=FALSE;
	xHardwareError:=FALSE;
	xQuitErr:=FALSE;
	xError:=FALSE;
	iErrorNr:=0;
	xInitError:=FALSE;
	xFreeze:=FALSE;
	xAbord:=FALSE;
	xReset:=FALSE;
	xCheckToolFeedPosition:=FALSE;
	bActivePartNumber:=0;
(*	lrProcessToolFeederActualPosition:=0.0;*)
	lrProcessToolFeederSpeed:=0.0;
	rSpeedToolFeed:=0.0;
	xCheckWithoutToolRotation:=FALSE;
END_IF;
END_FUNCTION_BLOCK

(* POU PRG_STATION_LAYER3/FB_STATIONEN/FB_FUNCTION/FB_FctToolCalibration, ST *)
FUNCTION_BLOCK FB_FctToolCalibration
VAR_INPUT
	xMicroRodActive: BOOL;		(* choice of the machine MicroWire or MicroRod *)
	xBeckhoffDriveActive: BOOL;	(* choice of the axis Beckhoff or EcoStep *)
	xSafetyCircuitOn:BOOL;			(* state of the safety circuit-->TRUE=Machine current ON, FALSE=Machine current OFF *)
	T_ProcessImageData:ST_RETAIN_DATA_PROCESSIMAGE;	(* Novram data structure for the process parameter *)
	T_Standard:ST_RETAIN_DATA;							(* Novram data structure for the standard process parameter *)
END_VAR
VAR_IN_OUT
	xStart : BOOL;					(* start the function *)
	xReset : BOOL;				(* reset the function *)
	xStop : BOOL;					(* stop the active function *)
	xQuitErr : BOOL;				(* quit the error caused of the active function *)
	xAbord : BOOL;				(* abord the active function *)
	TAxisToolLeft:ST_AXIS;		(* data structure for the ToolLeft axis *)
	TAxisToolCenter:ST_AXIS;		(* data structure for the ToolCenter axis *)
	TAxisToolRight:ST_AXIS;		(* data structure for the ToolRight axis *)
	TAxisToolFeeder:ST_AXIS;		(* data structure for the ToolFeeder axis *)
	TAxisGrindFeeder:ST_AXIS;	(* data structure for the GrindFeeder axis *)
	T_WorkTool:ST_WORKTOOL;	(* Tool parameter *)
END_VAR
VAR_OUTPUT
	xEnd : BOOL;					(* state of the function if a active function is ended *)
	xError : BOOL;					(* state of the function if a active function caused an error *)
	iErrorNr : INT;					(* state of the function if a active function caused an error, in this case give the error number *)
	lrProcessToolFeederActualPosition:LREAL;	(* gives the calculated position of the ToolFeeder *)
	lrProcessToolFeederSpeed:LREAL;			(* gives the calculated speed of the ToolFeeder *)
END_VAR
VAR
	xHardwareError: BOOL := FALSE;
	xInitError: BOOL := FALSE;
	iStepError: INT := 0;
	xStartMainCtr: BOOL := FALSE;
	xStartMainPrc: BOOL := FALSE;
	xInitMainCtr: BOOL := FALSE;
	iStepPrc: INT := 0;
	xSetEnd: BOOL := FALSE;
	xInitStep: BOOL := FALSE;
	xFreeze: BOOL := FALSE;
	iTmpErrorNr:INT:=0;
	xTmpInit:BOOL;
	iTmp:INT;
	xTmp: BOOL;
	xReadFirstTime: BOOL;
	xTmp1: BOOL;
	rToolRotationSpeed: REAL;
	FBToolCalcul:FB_TOOL_CALCUL_NEW;
	rToolFeedLength: REAL;
	rToolDiameter: REAL;
	rGrindFeedPlunge: REAL;
	ii: INT;
	iStartSection: INT;
	iEndSection: INT;
	rSpeedGrindFeed: REAL;
	rSpeedToolFeed: REAL;
	rTimeGrindPlunge: REAL;
	FBCalcGearFactor: FB_CALC_GEARFACTOR;
	lrToolFeederActualPosition: LREAL;
	iTmpStartSection: INT;
	FBCalcPlungeGrinding: FB_CALC_PLUNGE_GRINDING;
	xResetFB: BOOL;
	xGrindFeedMaster: BOOL;
	xCheckToolFeedPosition: BOOL;
	lrToolFeederPosition: LREAL;
	lrToolRightPosition: LREAL;
	lrSaveToolFeederPosition: LREAL;
	lrSaveToolRightPosition: LREAL;
	rPlungeCycleGrindFeedGeometry: REAL;
	lrToolFeedCalcLengthPosition: REAL;
	lrCalcToolLengthInc: LREAL;
	lrCalcToolLength: LREAL;
	rTimeToolFeed: REAL;
	xReadyToolFeedStop: BOOL;
	xReadyGrindFeedStop: BOOL;
END_VAR
(****************************************************************************************************************************************************)
(***********                                    This Functionblock define the function for the calibration of the tool                                            ************)
(****************************************************************************************************************************************************)

IF NOT(xReadFirstTime) THEN
	xReadFirstTime:=TRUE;
END_IF;
(******************************************************************************************************************************************)
(****************************				           Reset Function Part                                                 *****************************)
(******************************************************************************************************************************************)
IF xReset AND NOT(xSetEnd) THEN
	xEnd:=FALSE;
	xSetEnd:=TRUE;
END_IF;
(******************************************************************************************************************************************)
(****************************				              Error Controlling Part                                            *****************************)
(******************************************************************************************************************************************)
xTmp:=	TAxisToolLeft.T_CtrleSingle.xErr OR
		(TAxisToolCenter.T_CtrleSingle.xErr AND xMicroRodActive) OR
		TAxisToolRight.T_CtrleSingle.xErr OR
		TAxisToolFeeder.T_CtrleSingle.xErr OR
		TAxisGrindFeeder.T_CtrleSingle.xErr;
xTmp1:=	NOT(TAxisToolLeft.T_CtrleSingle.xExecute) AND
		((NOT(TAxisToolCenter.T_CtrleSingle.xExecute) AND xMicroRodActive) OR NOT(xMicroRodActive)) AND
		 NOT(TAxisToolRight.T_CtrleSingle.xExecute) AND
		((NOT(TAxisToolFeeder.T_CtrleSingle.xExecute) AND NOT(xMicroRodActive)) OR xMicroRodActive) AND
		NOT(TAxisGrindFeeder.T_CtrleSingle.xExecute);
IF (xHardwareError OR (xTmp AND xStartMainPrc)) AND NOT(xSetEnd) THEN
	IF xTmp1 THEN
		IF NOT(xInitError) THEN
			iStepError:=100;
			xInitError:=TRUE;
			IF xHardwareError THEN
				iErrorNr:=iTmpErrorNr;
			ELSE
				xHardwareError:=TRUE;	(* Hardware Error *)
			END_IF;
		END_IF;
		CASE iStepError OF
			100:	iStepError:=0;
				xError:=TRUE;
		END_CASE;
		IF xQuitErr THEN
			xSetEnd:=TRUE;
		END_IF;
	END_IF;
END_IF;
(******************************************************************************************************************************************)
(****************************				              Main Controlling Part                                            *****************************)
(******************************************************************************************************************************************)
IF (xStart OR xStartMainCtr) AND NOT(xSetEnd) AND NOT(xHardwareError) THEN
	IF NOT (xInitMainCtr) THEN
		iTmpErrorNr:=0;
		iStepPrc:=100;
		xInitMainCtr:=TRUE;
		xStartMainCtr:=TRUE;
		xStart:=FALSE;
		xEnd:=FALSE;
		xAbord:=FALSE;
		xTmpInit:=FALSE;
		xCheckToolFeedPosition:=FALSE;
		lrCalcToolLengthInc:=lrCalcToolLength:=0.0;
		rSpeedToolFeed:=0.0;
	END_IF;
	IF xStop AND NOT(xTmpInit) THEN
		xTmpInit:=TRUE;
		iTmp:=100;
		RETURN;
	END_IF;
	IF xFreeze THEN
		IF xStart AND NOT(xAbord) THEN
			xFreeze:=FALSE;
			xStart:=FALSE;
		END_IF;
		IF xAbord THEN
			xAbord:=FALSE;
			xFreeze:=FALSE;
			xStart:=FALSE;
			xSetEnd:=TRUE;
		END_IF;
		RETURN;
	END_IF;
	IF NOT(xStartMainPrc) AND NOT(xSetEnd) THEN
		xStartMainPrc:=TRUE;
	END_IF;
END_IF;
(******************************************************************************************************************************************)
(****************************		               Controlling of the ToolFeeder Position                            *****************************)
(******************************************************************************************************************************************)
IF xCheckToolFeedPosition THEN
	IF xMicroRodActive THEN
		lrToolFeederPosition:=TAxisToolFeeder.T_LiveValue.lrActualPositionNotModulo - lrSaveToolFeederPosition;
		lrToolFeederActualPosition:=(lrToolFeederPosition / TAxisToolFeeder.T_CtrleSingle.lrScaleFactor);
		lrCalcToolLength:=lrToolFeederActualPosition;
	END_IF;
	IF NOT(xMicroRodActive) AND (TAxisToolRight.T_CtrleSingle.lrGearRatio <> 0.0) THEN
		lrToolFeedCalcLengthPosition:=((((T_WorkTool.rToolLength * 10.0) / ABS(T_WorkTool.rPitch)) * 24000.0) / TAxisToolRight.T_CtrleSingle.lrScaleFactor);
		lrToolFeederPosition:=lrToolFeederPosition + ABS(ABS(TAxisToolRight.T_LiveValue.lrActualPosition) - (lrSaveToolFeederPosition / TAxisToolRight.T_CtrleSingle.lrScaleFactor));
		lrSaveToolFeederPosition:=ABS(TAxisToolRight.T_LiveValue.lrActualPositionNotModulo);
		lrToolFeederActualPosition:=((T_WorkTool.rToolLength * 10.0) / lrToolFeedCalcLengthPosition) * lrToolFeederPosition;
		lrCalcToolLength:=lrCalcToolLengthInc + lrToolFeederActualPosition;
	END_IF;
ELSE
	IF NOT(xMicroRodActive) AND (TAxisToolRight.T_CtrleSingle.lrGearRatio <> 0.0) THEN
		lrSaveToolFeederPosition:=ABS(TAxisToolRight.T_LiveValue.lrActualPositionNotModulo);
		lrSaveToolRightPosition:=TAxisToolRight.T_LiveValue.lrActualPositionNotModulo * TAxisToolRight.T_CtrleSingle.lrGearRatio;
		lrCalcToolLengthInc:=lrCalcToolLength;
	END_IF;
	IF xMicroRodActive THEN
		lrSaveToolFeederPosition:=TAxisToolFeeder.T_LiveValue.lrActualPositionNotModulo;
	END_IF;
	lrToolFeederActualPosition:=lrToolFeederPosition:=0.0;
END_IF;
lrProcessToolFeederActualPosition:=lrCalcToolLength;
lrProcessToolFeederSpeed:=rSpeedToolFeed;
(******************************************************************************************************************************************)
(****************************				             immediate Stop Part                                              *****************************)
(******************************************************************************************************************************************)
IF xTmpInit AND NOT(xSetEnd) THEN
	IF NOT(xSafetyCircuitOn) THEN
		xTmpInit:=FALSE;
		iTmp:=100;
		xSetEnd:=TRUE;
		RETURN;
	END_IF;
	CASE iTmp OF
		100:	xReadyToolFeedStop:=xReadyGrindFeedStop:=FALSE;
			TAxisGrindFeeder.T_CtrleSingle.lrAcceleration:=T_Standard.T_TeachINToolFeeder.rAcceleration;
			TAxisGrindFeeder.T_CtrleSingle.lrDecceleration:=T_Standard.T_TeachINToolFeeder.rDeceleration;
			TAxisGrindFeeder.T_CtrleSingle.iFunction:=5;	(* Stop Movement *)
			TAxisGrindFeeder.T_CtrleSingle.xExecute:=TRUE;
			iTmp:=200;
			RETURN;
		200:	IF NOT(TAxisGrindFeeder.T_CtrleSingle.xExecute) AND TAxisGrindFeeder.T_CtrleSingle.xDone THEN
				TAxisGrindFeeder.T_CtrleSingle.lrAcceleration:=T_Standard.T_TeachINGrindFeeder.rAcceleration;
				TAxisGrindFeeder.T_CtrleSingle.lrDecceleration:=T_Standard.T_TeachINGrindFeeder.rDeceleration;
				TAxisGrindFeeder.T_CtrleSingle.lrPosition:=	T_ProcessImageData.T_ProcessPara.rToolDiameterProcess +
														T_ProcessImageData.T_ProcessPara.rSecurityPosGrindFeedProcess;
				TAxisGrindFeeder.T_CtrleSingle.lrVelocity:=T_ProcessImageData.T_ProcessPara.rSpeedBackwardGrindFeed;
				TAxisGrindFeeder.T_CtrleSingle.iFunction:=7;	(* Move Absolut *)
				TAxisGrindFeeder.T_CtrleSingle.xExecute:=TRUE;
				iTmp:=300;
			END_IF;
			RETURN;
		300:	IF NOT(TAxisGrindFeeder.T_CtrleSingle.xExecute) AND TAxisGrindFeeder.T_CtrleSingle.xDone AND NOT(xReadyGrindFeedStop) THEN
				xReadyGrindFeedStop:=TRUE;
			END_IF;
			IF (TAxisGrindFeeder.T_LiveValue.lrActualPosition >= (T_ProcessImageData.T_ProcessPara.rToolDiameterProcess + T_ProcessImageData.T_ProcessPara.rOffsetBeforeToolDiaGrindFeedProcess)) AND NOT(xReadyToolFeedStop) THEN
				xReadyToolFeedStop:=TRUE;
				xCheckToolFeedPosition:=FALSE;
				IF xMicroRodActive THEN
					IF NOT(TAxisToolFeeder.T_CtrleSingle.xNotMoving) THEN
						TAxisToolFeeder.T_CtrleSingle.lrAcceleration:=T_Standard.T_TeachINToolFeeder.rAcceleration;
						TAxisToolFeeder.T_CtrleSingle.lrDecceleration:=T_Standard.T_TeachINToolFeeder.rDeceleration;
						TAxisToolFeeder.T_CtrleSingle.iFunction:=5;	(* Stop Movement *)
						TAxisToolFeeder.T_CtrleSingle.xExecute:=TRUE;
					END_IF;
				END_IF;
				IF NOT(xMicroRodActive) THEN
					FBCalcGearFactor(	rSpeed:= 0.0,
										rToolRotationSpeed:= rToolRotationSpeed,
										T_WorkTool:=T_WorkTool );
					TAxisToolFeeder.T_CtrleSingle.lrGearFactor:=INT_TO_LREAL(FBCalcGearFactor.T_WorkTool.iToolFeederGearFactor) * -1.0;
					TAxisToolFeeder.T_CtrleSingle.lrGearDivider:=INT_TO_LREAL(FBCalcGearFactor.T_WorkTool.iToolFeederGearDivider);
					(* Set Gear Value with PDO Object *)
					TAxisToolFeeder.T_RxPdoParameter.iGearFactor:=LREAL_TO_INT(TAxisToolFeeder.T_CtrleSingle.lrGearFactor);
					TAxisToolFeeder.T_RxPdoParameter.uiGearDivider:=LREAL_TO_UINT(TAxisToolFeeder.T_CtrleSingle.lrGearDivider);
				END_IF;
				lrProcessToolFeederSpeed:=0.0;
			END_IF;
			IF xReadyToolFeedStop AND xReadyGrindFeedStop THEN
				iTmp:=400;
			END_IF;
			RETURN;
		400:	IF NOT(TAxisToolFeeder.T_CtrleSingle.xExecute) AND TAxisToolFeeder.T_CtrleSingle.xDone THEN
				iTmp:=500;
			END_IF;
			RETURN;
		500:	xTmpInit:=FALSE;
			iTmp:=100;
			xSetEnd:=TRUE;
			RETURN;
	END_CASE;
END_IF;
(******************************************************************************************************************************************)
(****************************				             Main Procedure Part                                             *****************************)
(******************************************************************************************************************************************)
IF xStartMainPrc AND NOT(xSetEnd) AND NOT(xHardwareError) THEN
	CASE iStepPrc OF
		(* Initial Procedure *)
		100:	rToolFeedLength:=0.0;
			rToolDiameter:=T_ProcessImageData.T_ProcessPara.rToolDiameterProcess;
			rGrindFeedPlunge:=0.0;
			rSpeedGrindFeed:=0.0;
			rSpeedToolFeed:=0.0;
			xStartMainPrc:=FALSE;
			xInitStep:=FALSE;
			iStepPrc:=200;
		(* Calculation first only for the Plunge Procedure *)
		200:	IF NOT(xInitStep) THEN
				xInitStep:=TRUE;
				rToolFeedLength:=0.0;
				rSpeedToolFeed:=0.0;
				IF T_ProcessImageData.T_CalibrationPara.xPlungeActivationCalib THEN
					rToolFeedLength:=T_ProcessImageData.T_CalibrationPara.rPlungeLengthToolFeedCalib;
					T_WorkTool.rToolLength:=rToolFeedLength/10.0;
				ELSE
					T_WorkTool.rToolLength:=0.0;
				END_IF;
				IF T_ProcessImageData.T_CalibrationPara.xPlungeActivationCalib THEN
					T_WorkTool.rToolRotationSpeed:=T_ProcessImageData.T_CalibrationPara.rSpeedToolRotationCalib;
					T_WorkTool.rPitch:=T_ProcessImageData.T_CalibrationPara.rPitchCalib * -1.0;
					T_WorkTool.rGrindFeederPlunge:=	T_ProcessImageData.T_ProcessPara.rOffsetBeforeToolDiaGrindFeedProcess;
					FBToolCalcul(	xMicroRodActive:=xMicroRodActive,
									xBeckhoffDriveActive:=FALSE,
									T_WorkTool:= T_WorkTool,
									rToolFeedAcclDecl:= T_Standard.T_TeachINToolFeeder.rAcceleration);
					rGrindFeedPlunge:=T_WorkTool.rGrindFeederPlunge * -1.0;
					rSpeedGrindFeed:=T_WorkTool.rGrindFeederSpeedUnit;
					rSpeedToolFeed:=T_WorkTool.rToolFeederSpeedUnit * -1.0;
				ELSE
					rSpeedGrindFeed:=T_ProcessImageData.T_CalibrationPara.rPlungeSpeedGrindFeedCalib;
					rGrindFeedPlunge:=T_ProcessImageData.T_ProcessPara.rOffsetBeforeToolDiaGrindFeedProcess * -1.0;
					IF (rToolFeedLength <> 0) THEN
						rTimeGrindPlunge:=ABS(rGrindFeedPlunge) / rSpeedGrindFeed;		(* calc Time in seocnds *)
						rSpeedToolFeed:=rToolFeedLength / rTimeGrindPlunge;	(* calc Speed ToolFeed in mm/s *)
					END_IF;
					T_WorkTool.rPitch:=T_ProcessImageData.T_CalibrationPara.rPitchCalib * -1.0;
				END_IF;
				rToolRotationSpeed:=T_ProcessImageData.T_CalibrationPara.rSpeedToolRotationCalib;
				(* Start Relative movement of the GrindAxis *)
				TAxisGrindFeeder.T_CtrleSingle.lrAcceleration:=T_Standard.T_TeachINGrindFeeder.rAcceleration;
				TAxisGrindFeeder.T_CtrleSingle.lrDecceleration:=T_Standard.T_TeachINGrindFeeder.rDeceleration;
				TAxisGrindFeeder.T_CtrleSingle.lrDistance:=rGrindFeedPlunge;
				TAxisGrindFeeder.T_CtrleSingle.lrVelocity:=rSpeedGrindFeed;
				TAxisGrindFeeder.T_CtrleSingle.iFunction:=8;	(* Move Relative *)
				TAxisGrindFeeder.T_CtrleSingle.xExecute:=TRUE;
				IF (rToolFeedLength <> 0) THEN
					IF xMicroRodActive THEN
						(* Start continuos movement of the ToolFeeder Axis *)
						TAxisToolFeeder.T_CtrleSingle.lrAcceleration:=T_Standard.T_TeachINToolFeeder.rAcceleration;
						TAxisToolFeeder.T_CtrleSingle.lrDecceleration:=T_Standard.T_TeachINToolFeeder.rDeceleration;
						TAxisToolFeeder.T_CtrleSingle.lrVelocity:=rSpeedToolFeed;
						TAxisToolFeeder.T_CtrleSingle.iFunction:=6;	(* Move continue velocity *)
						TAxisToolFeeder.T_CtrleSingle.xExecute:=TRUE;
					ELSE
						FBCalcGearFactor(	rSpeed:= rSpeedToolFeed * -1.0,
											rToolRotationSpeed:= rToolRotationSpeed,
											T_WorkTool:=T_WorkTool );
						TAxisToolFeeder.T_CtrleSingle.lrGearFactor:=INT_TO_LREAL(FBCalcGearFactor.T_WorkTool.iToolFeederGearFactor) * -1.0;
						TAxisToolFeeder.T_CtrleSingle.lrGearDivider:=INT_TO_LREAL(FBCalcGearFactor.T_WorkTool.iToolFeederGearDivider);
						(* Set Gear Value with PDO Object *)
						TAxisToolFeeder.T_RxPdoParameter.iGearFactor:=LREAL_TO_INT(TAxisToolFeeder.T_CtrleSingle.lrGearFactor);
						TAxisToolFeeder.T_RxPdoParameter.uiGearDivider:=LREAL_TO_UINT(TAxisToolFeeder.T_CtrleSingle.lrGearDivider);
					END_IF;
				END_IF;
				IF (rToolFeedLength <> 0) THEN
					xCheckToolFeedPosition:=TRUE;	(* Start Measure Relative Position of the ToolFeeder *)
				END_IF;
			END_IF;
			IF NOT(TAxisGrindFeeder.T_CtrleSingle.xExecute) AND TAxisGrindFeeder.T_CtrleSingle.xDone THEN
				xCheckToolFeedPosition:=FALSE;
				xStartMainPrc:=FALSE;
				xInitStep:=FALSE;
				iStepPrc:=300;
			END_IF;
		(* Work the cylinder Part for the ToolCalibration *)
		300:	IF NOT(xInitStep) THEN
				xInitStep:=TRUE;
				T_WorkTool.rToolRotationSpeed:=T_ProcessImageData.T_CalibrationPara.rSpeedToolRotationCalib;
				T_WorkTool.rPitch:=T_ProcessImageData.T_CalibrationPara.rPitchCalib * -1.0;
				T_WorkTool.rToolLength:=T_ProcessImageData.T_CalibrationPara.rToolLengthCylinderPartCalib;
				rGrindFeedPlunge:=0.0;
				T_WorkTool.rGrindFeederPlunge:=0.0;
				FBToolCalcul(	xMicroRodActive:=xMicroRodActive,
								xBeckhoffDriveActive:=FALSE,
								T_WorkTool:= T_WorkTool,
								rToolFeedAcclDecl:= 0);
				rSpeedGrindFeed:=0.0;
				rToolFeedLength:=T_WorkTool.rToolLength;
				rSpeedToolFeed:=T_WorkTool.rToolFeederSpeedUnit;
				rToolRotationSpeed:=T_WorkTool.rToolRotationSpeed;
				IF xMicroRodActive THEN
					(* Start continuos movement of the ToolFeeder Axis *)
					TAxisToolFeeder.T_CtrleSingle.lrAcceleration:=T_Standard.T_TeachINToolFeeder.rAcceleration;
					TAxisToolFeeder.T_CtrleSingle.lrDecceleration:=T_Standard.T_TeachINToolFeeder.rDeceleration;
					TAxisToolFeeder.T_CtrleSingle.lrVelocity:=rSpeedToolFeed * -1.0;
					TAxisToolFeeder.T_CtrleSingle.iFunction:=6;	(* Move continue velocity *)
					TAxisToolFeeder.T_CtrleSingle.xExecute:=TRUE;
				ELSE
					TAxisToolFeeder.T_CtrleSingle.lrGearFactor:=INT_TO_LREAL(T_WorkTool.iToolFeederGearFactor) * -1.0;
					TAxisToolFeeder.T_CtrleSingle.lrGearDivider:=INT_TO_LREAL(T_WorkTool.iToolFeederGearDivider);
					(* Set Gear Value with PDO Object *)
					TAxisToolFeeder.T_RxPdoParameter.iGearFactor:=LREAL_TO_INT(TAxisToolFeeder.T_CtrleSingle.lrGearFactor);
					TAxisToolFeeder.T_RxPdoParameter.uiGearDivider:=LREAL_TO_UINT(TAxisToolFeeder.T_CtrleSingle.lrGearDivider);
				END_IF;
				xCheckToolFeedPosition:=TRUE;
				RETURN;
			END_IF;
			IF (lrToolFeederActualPosition > (rToolFeedLength * 10.0)) THEN
				xCheckToolFeedPosition:=FALSE;
				xStartMainPrc:=FALSE;
				xInitStep:=FALSE;
				iStepPrc:=400;
			END_IF;
		(* Displace Procedure Calculation *)
		400:IF NOT(xInitStep) THEN
				xInitStep:=TRUE;
				rToolFeedLength:=0.0;
				rSpeedToolFeed:=0.0;
				IF T_ProcessImageData.T_CalibrationPara.xDisplaceActivationCalib THEN
					rToolFeedLength:=T_ProcessImageData.T_CalibrationPara.rDisplaceLengthToolFeedCalib;
					T_WorkTool.rToolLength:=rToolFeedLength/10.0;
				ELSE
					T_WorkTool.rToolLength:=0.0;
				END_IF;
				IF T_ProcessImageData.T_CalibrationPara.xDisplaceActivationCalib THEN
					T_WorkTool.rToolRotationSpeed:=T_ProcessImageData.T_CalibrationPara.rSpeedToolRotationCalib;
					T_WorkTool.rPitch:=T_ProcessImageData.T_CalibrationPara.rPitchCalib * -1.0;
					T_WorkTool.rGrindFeederPlunge:=	T_ProcessImageData.T_ProcessPara.rOffsetBeforeToolDiaGrindFeedProcess;
					FBToolCalcul(	xMicroRodActive:=xMicroRodActive,
									xBeckhoffDriveActive:=FALSE,
									T_WorkTool:= T_WorkTool,
									rToolFeedAcclDecl:= T_Standard.T_TeachINToolFeeder.rDeceleration);
					rGrindFeedPlunge:=T_WorkTool.rGrindFeederPlunge;
					rSpeedGrindFeed:=T_WorkTool.rGrindFeederSpeedUnit;
					rSpeedToolFeed:=T_WorkTool.rToolFeederSpeedUnit * -1.0;
				ELSE
					rSpeedGrindFeed:=T_ProcessImageData.T_CalibrationPara.rDisplaceSpeedGrindFeedCalib;
					rGrindFeedPlunge:=T_ProcessImageData.T_ProcessPara.rOffsetBeforeToolDiaGrindFeedProcess;
					IF (rToolFeedLength <> 0) THEN
						rTimeGrindPlunge:=ABS(rGrindFeedPlunge) / rSpeedGrindFeed;		(* calc Time in seocnds *)
						rSpeedToolFeed:=(rToolFeedLength * 10.0) / rTimeGrindPlunge;	(* calc Speed ToolFeed in mm/s *)
					END_IF;
					T_WorkTool.rPitch:=T_ProcessImageData.T_CalibrationPara.rPitchCalib * -1.0;
				END_IF;
				rToolRotationSpeed:=T_ProcessImageData.T_CalibrationPara.rSpeedToolRotationCalib;
				(* Start Relative movement of the GrindAxis *)
				TAxisGrindFeeder.T_CtrleSingle.xBlockAcclDeclParameter:=TRUE;	(* do not send again the accl and decl parameter-->better performance *)
				TAxisGrindFeeder.T_CtrleSingle.lrAcceleration:=T_Standard.T_TeachINGrindFeeder.rAcceleration;
				TAxisGrindFeeder.T_CtrleSingle.lrDecceleration:=T_Standard.T_TeachINGrindFeeder.rDeceleration;
				TAxisGrindFeeder.T_CtrleSingle.lrDistance:=rGrindFeedPlunge;
				TAxisGrindFeeder.T_CtrleSingle.lrVelocity:=rSpeedGrindFeed;
				TAxisGrindFeeder.T_CtrleSingle.iFunction:=8;	(* Move Relative *)
				TAxisGrindFeeder.T_CtrleSingle.xExecute:=TRUE;
				IF (rToolFeedLength = 0) THEN
				(* Stop ToolFeeder Movement *)
					IF xMicroRodActive THEN
						TAxisToolFeeder.T_CtrleSingle.lrAcceleration:=T_Standard.T_TeachINToolFeeder.rAcceleration;
						TAxisToolFeeder.T_CtrleSingle.lrDecceleration:=T_Standard.T_TeachINToolFeeder.rDeceleration;
						TAxisToolFeeder.T_CtrleSingle.iFunction:=5;	(* Stop Movement *)
						TAxisToolFeeder.T_CtrleSingle.xExecute:=TRUE;
					END_IF;
					IF NOT(xMicroRodActive) THEN
						FBCalcGearFactor(	rSpeed:= 0.0,
											rToolRotationSpeed:= rToolRotationSpeed,
											T_WorkTool:=T_WorkTool );
						TAxisToolFeeder.T_CtrleSingle.lrGearFactor:=(INT_TO_LREAL(FBCalcGearFactor.T_WorkTool.iToolFeederGearFactor) * -1.0);
						TAxisToolFeeder.T_CtrleSingle.lrGearDivider:=INT_TO_LREAL(FBCalcGearFactor.T_WorkTool.iToolFeederGearDivider);
						(* Set Gear Value with PDO Object *)
						TAxisToolFeeder.T_RxPdoParameter.iGearFactor:=LREAL_TO_INT(TAxisToolFeeder.T_CtrleSingle.lrGearFactor);
						TAxisToolFeeder.T_RxPdoParameter.uiGearDivider:=LREAL_TO_UINT(TAxisToolFeeder.T_CtrleSingle.lrGearDivider);
					END_IF;
				ELSE
					IF xMicroRodActive THEN
						(* Start continuos movement of the ToolFeeder Axis *)
						TAxisToolFeeder.T_CtrleSingle.lrAcceleration:=T_Standard.T_TeachINToolFeeder.rAcceleration;
						TAxisToolFeeder.T_CtrleSingle.lrDecceleration:=T_Standard.T_TeachINToolFeeder.rDeceleration;
						TAxisToolFeeder.T_CtrleSingle.lrVelocity:=rSpeedToolFeed;
						TAxisToolFeeder.T_CtrleSingle.iFunction:=6;	(* Move continue velocity *)
						TAxisToolFeeder.T_CtrleSingle.xExecute:=TRUE;
					ELSE
						FBCalcGearFactor(	rSpeed:= rSpeedToolFeed * -1.0,
											rToolRotationSpeed:= rToolRotationSpeed,
											T_WorkTool:=T_WorkTool );
						TAxisToolFeeder.T_CtrleSingle.lrGearFactor:=INT_TO_LREAL(FBCalcGearFactor.T_WorkTool.iToolFeederGearFactor) * -1.0;
						TAxisToolFeeder.T_CtrleSingle.lrGearDivider:=INT_TO_LREAL(FBCalcGearFactor.T_WorkTool.iToolFeederGearDivider);
						(* Set Gear Value with PDO Object *)
						TAxisToolFeeder.T_RxPdoParameter.iGearFactor:=LREAL_TO_INT(TAxisToolFeeder.T_CtrleSingle.lrGearFactor);
						TAxisToolFeeder.T_RxPdoParameter.uiGearDivider:=LREAL_TO_UINT(TAxisToolFeeder.T_CtrleSingle.lrGearDivider);
					END_IF;
				END_IF;
				IF (rToolFeedLength <> 0) THEN
					xCheckToolFeedPosition:=TRUE;	(* Start Measure Relative Position of the ToolFeeder *)
				END_IF;
			END_IF;
			IF NOT(TAxisGrindFeeder.T_CtrleSingle.xExecute) AND TAxisGrindFeeder.T_CtrleSingle.xDone THEN
				xCheckToolFeedPosition:=FALSE;
				xStartMainPrc:=FALSE;
				xInitStep:=FALSE;
				iStepPrc:=500;
			END_IF;
		(* Check if ToolFeeder Moves and stop it if it moves *)
		500:IF NOT(xInitStep) THEN
				xInitStep:=TRUE;
				IF (rToolFeedLength <> 0) THEN
				(* Stop ToolFeeder Movement *)
					IF xMicroRodActive THEN
						TAxisToolFeeder.T_CtrleSingle.lrAcceleration:=T_Standard.T_TeachINToolFeeder.rAcceleration;
						TAxisToolFeeder.T_CtrleSingle.lrDecceleration:=T_Standard.T_TeachINToolFeeder.rDeceleration;
						TAxisToolFeeder.T_CtrleSingle.iFunction:=5;	(* Stop Movement *)
						TAxisToolFeeder.T_CtrleSingle.xExecute:=TRUE;
					END_IF;
					IF NOT(xMicroRodActive) THEN
						FBCalcGearFactor(	rSpeed:= 0.0,
											rToolRotationSpeed:= rToolRotationSpeed,
											T_WorkTool:=T_WorkTool );
						TAxisToolFeeder.T_CtrleSingle.lrGearFactor:=(INT_TO_LREAL(FBCalcGearFactor.T_WorkTool.iToolFeederGearFactor) * -1.0);
						TAxisToolFeeder.T_CtrleSingle.lrGearDivider:=INT_TO_LREAL(FBCalcGearFactor.T_WorkTool.iToolFeederGearDivider);
						(* Set Gear Value with PDO Object *)
						TAxisToolFeeder.T_RxPdoParameter.iGearFactor:=LREAL_TO_INT(TAxisToolFeeder.T_CtrleSingle.lrGearFactor);
						TAxisToolFeeder.T_RxPdoParameter.uiGearDivider:=LREAL_TO_UINT(TAxisToolFeeder.T_CtrleSingle.lrGearDivider);
					END_IF;
				END_IF;
			END_IF;
			IF NOT(TAxisToolFeeder.T_CtrleSingle.xExecute) AND TAxisToolFeeder.T_CtrleSingle.xDone THEN
				xStartMainPrc:=FALSE;
				xInitStep:=FALSE;
				iStepPrc:=600;
			END_IF;
		(* GrindFeeder go to Security Position *)
		600:IF NOT(xInitStep) THEN
				xInitStep:=TRUE;
				TAxisGrindFeeder.T_CtrleSingle.lrAcceleration:=T_Standard.T_TeachINGrindFeeder.rAcceleration;
				TAxisGrindFeeder.T_CtrleSingle.lrDecceleration:=T_Standard.T_TeachINGrindFeeder.rDeceleration;
				TAxisGrindFeeder.T_CtrleSingle.lrPosition:=	T_ProcessImageData.T_ProcessPara.rToolDiameterProcess +
														T_ProcessImageData.T_ProcessPara.rSecurityPosGrindFeedProcess;
				TAxisGrindFeeder.T_CtrleSingle.lrVelocity:=T_ProcessImageData.T_ProcessPara.rSpeedBackwardGrindFeed;
				TAxisGrindFeeder.T_CtrleSingle.iFunction:=7;	(* Move Absolut *)
				TAxisGrindFeeder.T_CtrleSingle.xExecute:=TRUE;
			END_IF;
			IF NOT(TAxisGrindFeeder.T_CtrleSingle.xExecute) AND TAxisGrindFeeder.T_CtrleSingle.xDone THEN
				xStartMainPrc:=FALSE;
				xInitStep:=FALSE;
				iStepPrc:=700;
			END_IF;
		(* Set ToolFeeder to Measure Position *)
		700:IF NOT(xInitStep) THEN
				xInitStep:=TRUE;
				rToolFeedLength:=0.0;
				T_WorkTool.rToolLength:=(T_ProcessImageData.T_CalibrationPara.rMeasureOffsetToolFeedCalib / 10.0);
				rSpeedToolFeed:=T_ProcessImageData.T_ProcessPara.rSpeedForwardSlowGrindFeed;
				rToolRotationSpeed:=T_ProcessImageData.T_CalibrationPara.rSpeedToolRotationCalib;
				rTimeToolFeed:=(T_WorkTool.rToolLength * 10.0) / rSpeedToolFeed;		(* calc Time in seocnds *)
				T_WorkTool.rPitch:=(T_WorkTool.rToolLength * 10.0) / ((rToolRotationSpeed/60.0) * rTimeToolFeed);
				IF xMicroRodActive THEN
					TAxisToolFeeder.T_CtrleSingle.lrAcceleration:=T_Standard.T_TeachINToolFeeder.rAcceleration;
					TAxisToolFeeder.T_CtrleSingle.lrDecceleration:=T_Standard.T_TeachINToolFeeder.rDeceleration;
					TAxisToolFeeder.T_CtrleSingle.lrPosition:=T_ProcessImageData.T_CalibrationPara.rMeasurePosToolFeedCalib;
					TAxisToolFeeder.T_CtrleSingle.iFunction:=7;	(* Move Absolut *)
					TAxisToolFeeder.T_CtrleSingle.lrVelocity:=rSpeedToolFeed;
					TAxisToolFeeder.T_CtrleSingle.xExecute:=TRUE;
				ELSE
					FBCalcGearFactor(	rSpeed:= T_ProcessImageData.T_ProcessPara.rSpeedForwardSlowGrindFeed * -1.0,
										rToolRotationSpeed:= rToolRotationSpeed,
										T_WorkTool:=T_WorkTool );
					TAxisToolFeeder.T_CtrleSingle.lrGearFactor:=INT_TO_LREAL(FBCalcGearFactor.T_WorkTool.iToolFeederGearFactor) * -1.0;
					TAxisToolFeeder.T_CtrleSingle.lrGearDivider:=INT_TO_LREAL(FBCalcGearFactor.T_WorkTool.iToolFeederGearDivider);
					(* Set Gear Value with PDO Object *)
					TAxisToolFeeder.T_RxPdoParameter.iGearFactor:=LREAL_TO_INT(TAxisToolFeeder.T_CtrleSingle.lrGearFactor);
					TAxisToolFeeder.T_RxPdoParameter.uiGearDivider:=LREAL_TO_UINT(TAxisToolFeeder.T_CtrleSingle.lrGearDivider);
					xCheckToolFeedPosition:=TRUE;
					RETURN;
				END_IF;

			END_IF;
			IF xMicroRodActive THEN
				IF NOT(TAxisToolFeeder.T_CtrleSingle.xExecute) AND TAxisToolFeeder.T_CtrleSingle.xDone THEN
					(* Procedure is finished *)
					xStartMainPrc:=FALSE;
					xInitStep:=FALSE;
					iStepPrc:=0;
					xSetEnd:=TRUE;
				END_IF;
			END_IF;
			IF NOT(xMicroRodActive) THEN
				IF (lrToolFeederActualPosition > T_ProcessImageData.T_CalibrationPara.rMeasureOffsetToolFeedCalib) THEN
					FBCalcGearFactor(	rSpeed:= 0.0,
										rToolRotationSpeed:= rToolRotationSpeed,
										T_WorkTool:=T_WorkTool );
					TAxisToolFeeder.T_CtrleSingle.lrGearFactor:=(INT_TO_LREAL(FBCalcGearFactor.T_WorkTool.iToolFeederGearFactor) * -1.0);
					TAxisToolFeeder.T_CtrleSingle.lrGearDivider:=INT_TO_LREAL(FBCalcGearFactor.T_WorkTool.iToolFeederGearDivider);
					(* Set Gear Value with PDO Object *)
					TAxisToolFeeder.T_RxPdoParameter.iGearFactor:=LREAL_TO_INT(TAxisToolFeeder.T_CtrleSingle.lrGearFactor);
					TAxisToolFeeder.T_RxPdoParameter.uiGearDivider:=LREAL_TO_UINT(TAxisToolFeeder.T_CtrleSingle.lrGearDivider);
					xCheckToolFeedPosition:=FALSE;
					(* Procedure is finished *)
					xStartMainPrc:=FALSE;
					xInitStep:=FALSE;
					iStepPrc:=0;
					xSetEnd:=TRUE;
				END_IF;
			END_IF;
	END_CASE;
END_IF;
(******************************************************************************************************************************************)
(****************************				           Parallel Procedure Part                                          *****************************)
(******************************************************************************************************************************************)
(******************************************************************************************************************************************)
(****************************				             	Init / Reset Part                                                   *****************************)
(******************************************************************************************************************************************)
IF xSetEnd THEN
	xEnd:=TRUE;
	xInitStep:=FALSE;
	xSetEnd:=FALSE;
	xStop:=FALSE;
	xStartMainPrc:=FALSE;
	xInitMainCtr:=FALSE;
	xStartMainCtr:=FALSE;
	xStart:=FALSE;
	xHardwareError:=FALSE;
	xQuitErr:=FALSE;
	xError:=FALSE;
	iErrorNr:=0;
	xInitError:=FALSE;
	xFreeze:=FALSE;
	xAbord:=FALSE;
	xReset:=FALSE;
	xCheckToolFeedPosition:=FALSE;
(*	lrProcessToolFeederActualPosition:=0.0;*)
	lrProcessToolFeederSpeed:=0.0;
	rSpeedToolFeed:=0.0;
END_IF;
END_FUNCTION_BLOCK

(* POU PRG_STATION_LAYER3/FB_STATIONEN/FB_FUNCTION/FB_FctToolFeedAbsRelPosition, ST *)
FUNCTION_BLOCK FB_FctToolFeedAbsRelPosition
VAR_INPUT
	xMicroRodActive: BOOL;		(* choice of the machine MicroWire or MicroRod *)
	xBeckhoffDriveActive: BOOL;	(* choice of the axis Beckhoff or EcoStep *)
	xSafetyCircuitOn:BOOL;			(* state of the safety circuit-->TRUE=Machine current ON, FALSE=Machine current OFF *)
	iFunctionNr:INT;				(* state of the called function number-->14=move axis absolut, 15=move axis relative *)
END_VAR
VAR_IN_OUT
	xStart : BOOL;					(* start the function *)
	xReset : BOOL;				(* reset the function *)
	xStop : BOOL;					(* stop the active function *)
	xQuitErr : BOOL;				(* quit the error caused of the active function *)
	xAbord : BOOL;				(* abord the active function *)
	TAxisToolFeeder:ST_AXIS;		(* data structure for the ToolFeeder axis *)
END_VAR
VAR_OUTPUT
	xEnd : BOOL;					(* state of the function if a active function is ended *)
	xError : BOOL;					(* state of the function if a active function caused an error *)
	iErrorNr : INT;					(* state of the function if a active function caused an error, in this case give the error number *)
END_VAR
VAR
	xHardwareError: BOOL := FALSE;
	xInitError: BOOL := FALSE;
	iStepError: INT := 0;
	xStartMainCtr: BOOL := FALSE;
	xStartMainPrc: BOOL := FALSE;
	xInitMainCtr: BOOL := FALSE;
	iStepPrc: INT := 0;
	xSetEnd: BOOL := FALSE;
	xInitStep: BOOL := FALSE;
	xFreeze: BOOL := FALSE;
	iTmpErrorNr:INT:=0;
	xTmpInit:BOOL;
	iTmp:INT;
END_VAR
(****************************************************************************************************************************************************)
(***********       This Functionblock define the function for set the ToolFeeder Axis to the relative or absolut position         ************)
(****************************************************************************************************************************************************)

(******************************************************************************************************************************************)
(****************************				           Reset Function Part                                                 *****************************)
(******************************************************************************************************************************************)
IF xReset AND NOT(xSetEnd) THEN
	xEnd:=FALSE;
	xSetEnd:=TRUE;
END_IF;
(******************************************************************************************************************************************)
(****************************				              Error Controlling Part                                            *****************************)
(******************************************************************************************************************************************)
IF (xHardwareError OR ((TAxisToolFeeder.T_CtrleSingle.xErr) AND xStartMainPrc)) AND NOT(xSetEnd) THEN
	IF NOT(TAxisToolFeeder.T_CtrleSingle.xExecute) THEN
		IF NOT(xInitError) THEN
			iStepError:=100;
			xInitError:=TRUE;
			IF xHardwareError THEN
				iErrorNr:=iTmpErrorNr;
			ELSE
				xHardwareError:=TRUE;	(* Hardware Error *)
			END_IF;
		END_IF;
		CASE iStepError OF
			100:	iStepError:=0;
				xError:=TRUE;
		END_CASE;
		IF xQuitErr THEN
			xSetEnd:=TRUE;
		END_IF;
	END_IF;
END_IF;
(******************************************************************************************************************************************)
(****************************				              Main Controlling Part                                            *****************************)
(******************************************************************************************************************************************)
IF (xStart OR xStartMainCtr) AND NOT(xSetEnd) AND NOT(xHardwareError) THEN
	IF NOT (xInitMainCtr) THEN
		iTmpErrorNr:=0;
		iStepPrc:=100;
		xInitMainCtr:=TRUE;
		xStartMainCtr:=TRUE;
		xStart:=FALSE;
		xEnd:=FALSE;
		xAbord:=FALSE;
		xTmpInit:=FALSE;
	END_IF;
	IF xStop AND NOT(xTmpInit) THEN
		xTmpInit:=TRUE;
		iTmp:=100;
		RETURN;
	END_IF;
	IF xFreeze THEN
		IF xStart AND NOT(xAbord) THEN
			xFreeze:=FALSE;
			xStart:=FALSE;
		END_IF;
		IF xAbord THEN
			xAbord:=FALSE;
			xFreeze:=FALSE;
			xStart:=FALSE;
			xSetEnd:=TRUE;
		END_IF;
		RETURN;
	END_IF;
	IF NOT(xStartMainPrc) AND NOT(xSetEnd) THEN
		xStartMainPrc:=TRUE;
	END_IF;
END_IF;
(******************************************************************************************************************************************)
(****************************				             immediate Stop Part                                              *****************************)
(******************************************************************************************************************************************)
IF xTmpInit AND NOT(xSetEnd) THEN
	IF NOT(xSafetyCircuitOn) THEN
		xTmpInit:=FALSE;
		iTmp:=100;
		xSetEnd:=TRUE;
		RETURN;
	END_IF;
	CASE iTmp OF
		100:	TAxisToolFeeder.T_CtrleSingle.iFunction:=5;
			TAxisToolFeeder.T_CtrleSingle.xExecute:=TRUE;
			iTmp:=200;
			RETURN;
		200:	IF NOT(TAxisToolFeeder.T_CtrleSingle.xExecute) AND TAxisToolFeeder.T_CtrleSingle.xDone THEN
				iTmp:=300;
			END_IF;
			RETURN;
		300:	xTmpInit:=FALSE;
			iTmp:=100;
			xSetEnd:=TRUE;
			RETURN;
	END_CASE;
END_IF;
(******************************************************************************************************************************************)
(****************************				             Main Procedure Part                                             *****************************)
(******************************************************************************************************************************************)
IF xStartMainPrc AND NOT(xSetEnd) AND NOT(xHardwareError) THEN
	CASE iStepPrc OF
		100:	IF NOT(xInitStep) THEN
				xInitStep:=TRUE;
				IF NOT(TAxisToolFeeder.T_CtrleSingle.xDone)THEN
					xHardwareError:=TRUE;
					iTmpErrorNr:=1;
					RETURN;
				END_IF;
				IF NOT(TAxisToolFeeder.T_CtrleSingle.xPower) THEN
					TAxisToolFeeder.T_CtrleSingle.iFunction:=3;
					TAxisToolFeeder.T_CtrleSingle.xExecute:=TRUE;
				END_IF;
			END_IF;
			IF NOT(TAxisToolFeeder.T_CtrleSingle.xExecute) AND TAxisToolFeeder.T_CtrleSingle.xDone THEN
				xStartMainPrc:=FALSE;
				xInitStep:=FALSE;
				iStepPrc:=200;
			END_IF;
		200:	IF NOT(xInitStep) THEN
				xInitStep:=TRUE;
				IF (iFunctionNr = 14) THEN
					TAxisToolFeeder.T_CtrleSingle.iFunction:=7;	(* Move Absolut *)
				END_IF;
				IF (iFunctionNr = 15) THEN
					TAxisToolFeeder.T_CtrleSingle.iFunction:=8;	(* Move Relative *)
				END_IF;
				TAxisToolFeeder.T_CtrleSingle.xExecute:=TRUE;
			END_IF;
			IF NOT(TAxisToolFeeder.T_CtrleSingle.xExecute) AND TAxisToolFeeder.T_CtrleSingle.xDone THEN
				xStartMainPrc:=FALSE;
				xInitStep:=FALSE;
				iStepPrc:=0;
				xSetEnd:=TRUE;
			END_IF;
	END_CASE;
END_IF;
(******************************************************************************************************************************************)
(****************************				           Parallel Procedure Part                                          *****************************)
(******************************************************************************************************************************************)

(******************************************************************************************************************************************)
(****************************				             	Init / Reset Part                                                   *****************************)
(******************************************************************************************************************************************)
IF xSetEnd THEN
	xEnd:=TRUE;
	xInitStep:=FALSE;
	xSetEnd:=FALSE;
	xStop:=FALSE;
	xStartMainPrc:=FALSE;
	xInitMainCtr:=FALSE;
	xStartMainCtr:=FALSE;
	xStart:=FALSE;
	xHardwareError:=FALSE;
	xQuitErr:=FALSE;
	xError:=FALSE;
	iErrorNr:=0;
	xInitError:=FALSE;
	xFreeze:=FALSE;
	xAbord:=FALSE;
	xReset:=FALSE;
END_IF;
END_FUNCTION_BLOCK

(* POU PRG_STATION_LAYER3/FB_STATIONEN/FB_FUNCTION/FB_FctSwitchOnOffPowerSupply, ST *)
FUNCTION_BLOCK FB_FctSwitchOnOffPowerSupply
VAR_INPUT
	xMicroRodActive: BOOL;		(* choice of the machine MicroWire or MicroRod *)
	xBeckhoffDriveActive: BOOL;	(* choice of the axis Beckhoff or EcoStep *)
	xSafetyCircuitOn:BOOL;			(* state of the safety circuit-->TRUE=Machine current ON, FALSE=Machine current OFF *)
	iFunctionNr:INT;				(* state of the called function number-->16=switch current on of all axis, 17=switch current off of all axis *)
END_VAR
VAR_IN_OUT
	xStart : BOOL;					(* start the function *)
	xReset : BOOL;				(* reset the function *)
	xStop : BOOL;					(* stop the active function *)
	xQuitErr : BOOL;				(* quit the error caused of the active function *)
	xAbord : BOOL;				(* abord the active function *)
	TAxisToolLeft:ST_AXIS;		(* data structure for the ToolLeft axis *)
	TAxisToolCenter:ST_AXIS;		(* data structure for the ToolCenter axis *)
	TAxisToolRight:ST_AXIS;		(* data structure for the ToolRight axis *)
	TAxisToolFeeder:ST_AXIS;		(* data structure for the ToolFeeder axis *)
	TAxisGrindFeeder:ST_AXIS;	(* data structure for the GrindFeeder axis *)
	TAxisGrindSpindle:ST_AXIS;	(* data structure for the GrindSpindle axis *)			(* IGS *)
END_VAR
VAR_OUTPUT
	xEnd : BOOL;					(* state of the function if a active function is ended *)
	xError : BOOL;					(* state of the function if a active function caused an error *)
	iErrorNr : INT;					(* state of the function if a active function caused an error, in this case give the error number *)
END_VAR
VAR
	xHardwareError: BOOL := FALSE;
	xInitError: BOOL := FALSE;
	iStepError: INT := 0;
	xStartMainCtr: BOOL := FALSE;
	xStartMainPrc: BOOL := FALSE;
	xInitMainCtr: BOOL := FALSE;
	iStepPrc: INT := 0;
	xSetEnd: BOOL := FALSE;
	xInitStep: BOOL := FALSE;
	xFreeze: BOOL := FALSE;
	iTmpErrorNr:INT:=0;
	xTmpInit:BOOL;
	iTmp:INT;
	xTmp: BOOL;
	xTmp1: BOOL;
END_VAR
(****************************************************************************************************************************************************)
(***    This Functionblock switch the axis current on or off for the ToolLeft,ToolCenter,ToolRight,ToolFeeder or GrindFeeder     ***)
(****************************************************************************************************************************************************)

(******************************************************************************************************************************************)
(****************************				           Reset Function Part                                                 *****************************)
(******************************************************************************************************************************************)
IF xReset AND NOT(xSetEnd) THEN
	xEnd:=FALSE;
	xSetEnd:=TRUE;
END_IF;
(******************************************************************************************************************************************)
(****************************				              Error Controlling Part                                            *****************************)
(******************************************************************************************************************************************)
xTmp:=	TAxisToolLeft.T_CtrleSingle.xErr OR
		(TAxisToolCenter.T_CtrleSingle.xErr AND xMicroRodActive) OR
		TAxisToolRight.T_CtrleSingle.xErr OR
		TAxisToolFeeder.T_CtrleSingle.xErr OR
		TAxisGrindFeeder.T_CtrleSingle.xErr OR
		TAxisGrindSpindle.T_CtrleSingle.xErr;
xTmp1:=	NOT(TAxisToolLeft.T_CtrleSingle.xExecute) AND
		((NOT(TAxisToolCenter.T_CtrleSingle.xExecute) AND xMicroRodActive) OR NOT(xMicroRodActive)) AND
		 NOT(TAxisToolRight.T_CtrleSingle.xExecute) AND
		NOT(TAxisToolFeeder.T_CtrleSingle.xExecute) AND
		NOT(TAxisGrindFeeder.T_CtrleSingle.xExecute) AND
		NOT(TAxisGrindSpindle.T_CtrleSingle.xExecute);
IF (xHardwareError OR (xTmp AND xStartMainPrc)) AND NOT(xSetEnd) THEN
	IF xTmp1 THEN
		IF NOT(xInitError) THEN
			iStepError:=100;
			xInitError:=TRUE;
			IF xHardwareError THEN
				iErrorNr:=iTmpErrorNr;
			ELSE
				xHardwareError:=TRUE;	(* Hardware Error *)
			END_IF;
		END_IF;
		CASE iStepError OF
			100:	iStepError:=0;
				xError:=TRUE;
		END_CASE;
		IF xQuitErr THEN
			xSetEnd:=TRUE;
		END_IF;
	END_IF;
END_IF;
(******************************************************************************************************************************************)
(****************************				              Main Controlling Part                                            *****************************)
(******************************************************************************************************************************************)
IF (xStart OR xStartMainCtr) AND NOT(xSetEnd) AND NOT(xHardwareError) THEN
	IF NOT (xInitMainCtr) THEN
		iTmpErrorNr:=0;
		iStepPrc:=100;
		xInitMainCtr:=TRUE;
		xStartMainCtr:=TRUE;
		xStart:=FALSE;
		xEnd:=FALSE;
		xAbord:=FALSE;
		xTmpInit:=FALSE;
	END_IF;
	IF xStop AND NOT(xTmpInit) THEN
		xTmpInit:=TRUE;
		iTmp:=100;
		RETURN;
	END_IF;
	IF xFreeze THEN
		IF xStart AND NOT(xAbord) THEN
			xFreeze:=FALSE;
			xStart:=FALSE;
		END_IF;
		IF xAbord THEN
			xAbord:=FALSE;
			xFreeze:=FALSE;
			xStart:=FALSE;
			xSetEnd:=TRUE;
		END_IF;
		RETURN;
	END_IF;
	IF NOT(xStartMainPrc) AND NOT(xSetEnd) THEN
		xStartMainPrc:=TRUE;
	END_IF;
END_IF;
(******************************************************************************************************************************************)
(****************************				             immediate Stop Part                                              *****************************)
(******************************************************************************************************************************************)
IF xTmpInit AND NOT(xSetEnd) THEN
	IF NOT(xSafetyCircuitOn) THEN
		xTmpInit:=FALSE;
		iTmp:=100;
		xSetEnd:=TRUE;
		RETURN;
	END_IF;
	CASE iTmp OF
		100:	xTmp:=	NOT(TAxisToolLeft.T_CtrleSingle.xDone) OR
					(NOT(TAxisToolCenter.T_CtrleSingle.xDone) AND xMicroRodActive) OR
					NOT(TAxisToolRight.T_CtrleSingle.xDone) OR
					NOT(TAxisToolFeeder.T_CtrleSingle.xDone) OR
					NOT(TAxisGrindFeeder.T_CtrleSingle.xDone) OR
					NOT(TAxisGrindSpindle.T_CtrleSingle.xDone);
			IF xTmp THEN
				iTmp:=300;
				RETURN;
			END_IF;
			TAxisToolLeft.T_CtrleSingle.xReset:=NOT(TAxisToolLeft.T_CtrleSingle.xDone);
			TAxisToolCenter.T_CtrleSingle.xReset:=NOT(TAxisToolCenter.T_CtrleSingle.xDone) AND xMicroRodActive;
			TAxisToolRight.T_CtrleSingle.xReset:=NOT(TAxisToolRight.T_CtrleSingle.xDone);
			TAxisToolFeeder.T_CtrleSingle.xReset:=NOT(TAxisToolFeeder.T_CtrleSingle.xDone);
			TAxisGrindFeeder.T_CtrleSingle.xReset:=NOT(TAxisGrindFeeder.T_CtrleSingle.xDone);
			TAxisGrindSpindle.T_CtrleSingle.xReset:=NOT(TAxisGrindSpindle.T_CtrleSingle.xDone);
			iTmp:=200;
			RETURN;
		200:	xTmp:=	TAxisToolLeft.T_CtrleSingle.xDone AND
					((NOT(TAxisToolCenter.T_CtrleSingle.xDone) AND xMicroRodActive) OR NOT(xMicroRodActive)) AND
					TAxisToolRight.T_CtrleSingle.xDone AND
					TAxisToolFeeder.T_CtrleSingle.xDone AND
					TAxisGrindFeeder.T_CtrleSingle.xDone AND
					TAxisGrindSpindle.T_CtrleSingle.xDone;
			IF xTmp THEN
				iTmp:=300;
			END_IF;
			RETURN;
		300:	xTmpInit:=FALSE;
			iTmp:=100;
			xSetEnd:=TRUE;
			RETURN;
	END_CASE;
END_IF;
(******************************************************************************************************************************************)
(****************************				             Main Procedure Part                                             *****************************)
(******************************************************************************************************************************************)
IF xStartMainPrc AND NOT(xSetEnd) AND NOT(xHardwareError) THEN
	CASE iStepPrc OF
		100:	IF NOT(xInitStep) THEN
				xInitStep:=TRUE;
				xTmp:=	NOT(TAxisToolLeft.T_CtrleSingle.xDone) OR
						(NOT(TAxisToolCenter.T_CtrleSingle.xDone) AND xMicroRodActive) OR
						NOT(TAxisToolRight.T_CtrleSingle.xDone) OR
						NOT(TAxisToolFeeder.T_CtrleSingle.xDone) OR
						NOT(TAxisGrindFeeder.T_CtrleSingle.xDone) OR
						NOT(TAxisGrindSpindle.T_CtrleSingle.xDone);
				IF xTmp THEN
					xHardwareError:=TRUE;
					iTmpErrorNr:=1;
					RETURN;
				END_IF;
				IF (iFunctionNr = 16) THEN
				(* Switch On all Axis *)
					IF NOT(TAxisToolLeft.T_CtrleSingle.xPower) THEN
						TAxisToolLeft.T_CtrleSingle.iFunction:=3;
						TAxisToolLeft.T_CtrleSingle.xExecute:=TRUE;
					END_IF;
					IF xMicroRodActive THEN
						IF NOT(TAxisToolCenter.T_CtrleSingle.xPower) THEN
							TAxisToolCenter.T_CtrleSingle.iFunction:=3;
							TAxisToolCenter.T_CtrleSingle.xExecute:=TRUE;
						END_IF;
					END_IF;
					IF NOT(TAxisToolRight.T_CtrleSingle.xPower) THEN
						TAxisToolRight.T_CtrleSingle.iFunction:=3;
						TAxisToolRight.T_CtrleSingle.xExecute:=TRUE;
					END_IF;
					IF NOT(TAxisToolFeeder.T_CtrleSingle.xPower) THEN
						TAxisToolFeeder.T_CtrleSingle.iFunction:=3;
						TAxisToolFeeder.T_CtrleSingle.xExecute:=TRUE;
					END_IF;
					IF NOT(TAxisGrindFeeder.T_CtrleSingle.xPower) THEN
						TAxisGrindFeeder.T_CtrleSingle.iFunction:=3;
						TAxisGrindFeeder.T_CtrleSingle.xExecute:=TRUE;
					END_IF;
					IF NOT(TAxisGrindSpindle.T_CtrleSingle.xPower) THEN
						TAxisGrindSpindle.T_CtrleSingle.iFunction:=3;
						TAxisGrindSpindle.T_CtrleSingle.xExecute:=TRUE;
					END_IF;
				END_IF;
				IF (iFunctionNr = 17) THEN
				(* Switch Off all Axis *)
					IF TAxisToolLeft.T_CtrleSingle.xPower THEN
						TAxisToolLeft.T_CtrleSingle.iFunction:=4;
						TAxisToolLeft.T_CtrleSingle.xExecute:=TRUE;
					END_IF;
					IF xMicroRodActive THEN
						IF TAxisToolCenter.T_CtrleSingle.xPower THEN
							TAxisToolCenter.T_CtrleSingle.iFunction:=4;
							TAxisToolCenter.T_CtrleSingle.xExecute:=TRUE;
						END_IF;
					END_IF;
					IF TAxisToolRight.T_CtrleSingle.xPower THEN
						TAxisToolRight.T_CtrleSingle.iFunction:=4;
						TAxisToolRight.T_CtrleSingle.xExecute:=TRUE;
					END_IF;
					IF TAxisToolFeeder.T_CtrleSingle.xPower THEN
						TAxisToolFeeder.T_CtrleSingle.iFunction:=4;
						TAxisToolFeeder.T_CtrleSingle.xExecute:=TRUE;
					END_IF;
					IF TAxisGrindFeeder.T_CtrleSingle.xPower THEN
						TAxisGrindFeeder.T_CtrleSingle.iFunction:=4;
						TAxisGrindFeeder.T_CtrleSingle.xExecute:=TRUE;
					END_IF;
					IF TAxisGrindSpindle.T_CtrleSingle.xPower THEN
						TAxisGrindSpindle.T_CtrleSingle.iFunction:=4;
						TAxisGrindSpindle.T_CtrleSingle.xExecute:=TRUE;
					END_IF;
				END_IF;
			END_IF;
			IF NOT(TAxisToolLeft.T_CtrleSingle.xExecute) AND TAxisToolLeft.T_CtrleSingle.xDone AND
			    ((NOT(TAxisToolCenter.T_CtrleSingle.xExecute) AND TAxisToolCenter.T_CtrleSingle.xDone AND xMicroRodActive) OR NOT(xMicroRodActive)) AND
			    NOT(TAxisToolRight.T_CtrleSingle.xExecute) AND TAxisToolRight.T_CtrleSingle.xDone AND
			    NOT(TAxisToolFeeder.T_CtrleSingle.xExecute) AND TAxisToolFeeder.T_CtrleSingle.xDone AND
			    NOT(TAxisGrindFeeder.T_CtrleSingle.xExecute) AND TAxisGrindFeeder.T_CtrleSingle.xDone AND
			    NOT(TAxisGrindSpindle.T_CtrleSingle.xExecute) AND TAxisGrindSpindle.T_CtrleSingle.xDone THEN
				xStartMainPrc:=FALSE;
				xInitStep:=FALSE;
				iStepPrc:=0;
				xSetEnd:=TRUE;
			END_IF;
	END_CASE;
END_IF;
(******************************************************************************************************************************************)
(****************************				           Parallel Procedure Part                                          *****************************)
(******************************************************************************************************************************************)

(******************************************************************************************************************************************)
(****************************				             	Init / Reset Part                                                   *****************************)
(******************************************************************************************************************************************)
IF xSetEnd THEN
	xEnd:=TRUE;
	xInitStep:=FALSE;
	xSetEnd:=FALSE;
	xStop:=FALSE;
	xStartMainPrc:=FALSE;
	xInitMainCtr:=FALSE;
	xStartMainCtr:=FALSE;
	xStart:=FALSE;
	xHardwareError:=FALSE;
	xQuitErr:=FALSE;
	xError:=FALSE;
	iErrorNr:=0;
	xInitError:=FALSE;
	xFreeze:=FALSE;
	xAbord:=FALSE;
	xReset:=FALSE;
END_IF;
END_FUNCTION_BLOCK

(* POU PRG_STATION_LAYER3/FB_STATIONEN/FB_FUNCTION/FB_FctToolFeedMaxLenReference, ST *)
FUNCTION_BLOCK FB_FctToolFeedMaxLenReference
VAR_INPUT
	xMicroRodActive: BOOL;			(* choice of the machine MicroWire or MicroRod *)
	xBeckhoffDriveActive: BOOL;		(* choice of the axis Beckhoff or EcoStep *)
	xSafetyCircuitOn:BOOL;				(* state of the safety circuit-->TRUE=Machine current ON, FALSE=Machine current OFF *)
	T_Standard:ST_RETAIN_DATA;	(* Novram data structure for the standard process parameter *)
END_VAR
VAR_IN_OUT
	xStart : BOOL;					(* start the function *)
	xReset : BOOL;				(* reset the function *)
	xStop : BOOL;					(* stop the active function *)
	xQuitErr : BOOL;				(* quit the error caused of the active function *)
	xAbord : BOOL;				(* abord the active function *)
	TAxisToolFeeder:ST_AXIS;		(* data structure for the ToolFeeder axis *)
END_VAR
VAR_OUTPUT
	xEnd : BOOL;					(* state of the function if a active function is ended *)
	xError : BOOL;					(* state of the function if a active function caused an error *)
	iErrorNr : INT;					(* state of the function if a active function caused an error, in this case give the error number *)
END_VAR
VAR
	xHardwareError: BOOL := FALSE;
	xInitError: BOOL := FALSE;
	iStepError: INT := 0;
	xStartMainCtr: BOOL := FALSE;
	xStartMainPrc: BOOL := FALSE;
	xInitMainCtr: BOOL := FALSE;
	iStepPrc: INT := 0;
	xSetEnd: BOOL := FALSE;
	xInitStep: BOOL := FALSE;
	xFreeze: BOOL := FALSE;
	iTmpErrorNr:INT:=0;
	xTmpInit:BOOL;
	iTmp:INT;
	xToolFeederHWLimitPos: BOOL;
END_VAR
(****************************************************************************************************************************************************)
(*******                                This Functionblock define the function for reference the max length of the Tool (ToolFeeder Axis   ********)
(****************************************************************************************************************************************************)

